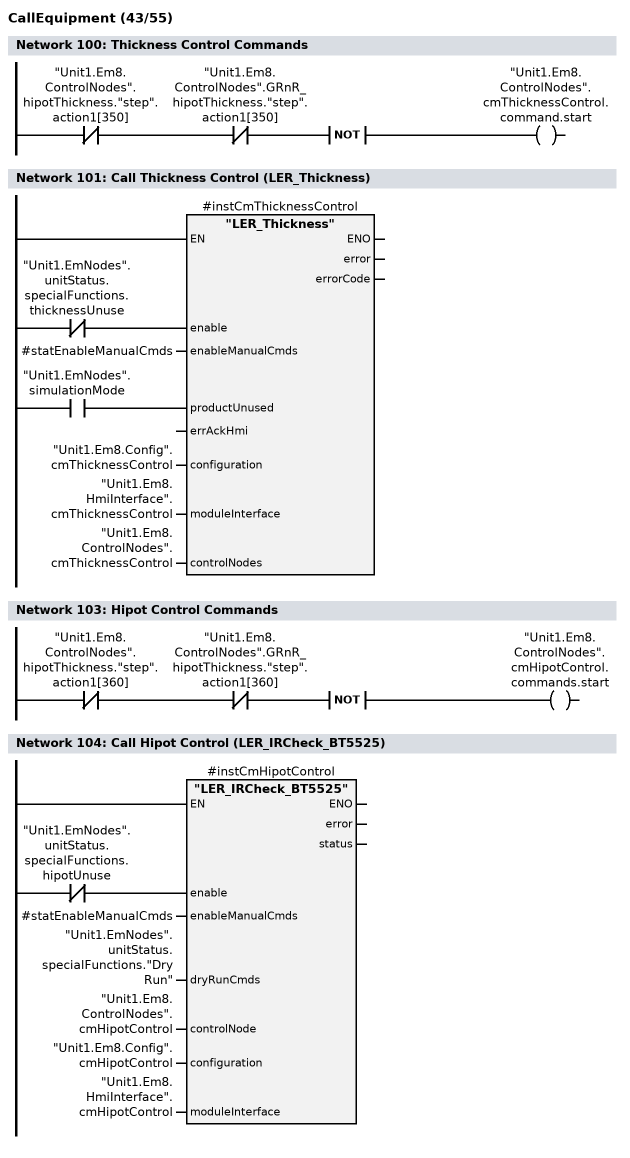
   RUNG wire#powerrail
      I_Contact( "Unit1.Em8.ControlNodes".hipotThickness."step".action1[350] )
      I_Contact( "Unit1.Em8.ControlNodes".GRnR_hipotThickness."step".action1[350] )
      Not()
      Coil( "Unit1.Em8.ControlNodes".cmThicknessControl.command.start )
   END_RUNG
   // the same network as SCL:
   "Unit1.Em8.ControlNodes".cmThicknessControl.command.start := NOT (NOT "Unit1.Em8.ControlNodes".hipotThickness."step".action1[350] AND NOT "Unit1.Em8.ControlNodes".GRnR_hipotThickness."step".action1[350]);
END_REGION

REGION Network 101: Call Thickness Control (LER_Thickness)
   RUNG wire#powerrail
      #instCmThicknessControl(enable := wire#w1, productUnused := wire#w2, enableManualCmds := #statEnableManualCmds, errAckHmi :=, configuration := "Unit1.Em8.Config".cmThicknessControl, moduleInterface := "Unit1.Em8.HmiInterface".cmThicknessControl, controlNodes := "Unit1.Em8.ControlNodes".cmThicknessControl, error =>, errorCode =>)
   END_RUNG
   RUNG wire#powerrail
      I_Contact( "Unit1.EmNodes".unitStatus.specialFunctions.thicknessUnuse )
   END_RUNG wire#w1
   RUNG wire#powerrail
      Contact( "Unit1.EmNodes".simulationMode )
   END_RUNG wire#w2
   // the same network as SCL:
   #instCmThicknessControl(enable := NOT "Unit1.EmNodes".unitStatus.specialFunctions.thicknessUnuse,   // "LER_Thickness"
                           enableManualCmds := #statEnableManualCmds,
                           productUnused := "Unit1.EmNodes".simulationMode,
                           configuration := "Unit1.Em8.Config".cmThicknessControl,
                           moduleInterface := "Unit1.Em8.HmiInterface".cmThicknessControl,
                           controlNodes := "Unit1.Em8.ControlNodes".cmThicknessControl);
END_REGION

REGION Network 103: Hipot Control Commands
   RUNG wire#powerrail
      I_Contact( "Unit1.Em8.ControlNodes".hipotThickness."step".action1[360] )
      I_Contact( "Unit1.Em8.ControlNodes".GRnR_hipotThickness."step".action1[360] )
      Not()
      Coil( "Unit1.Em8.ControlNodes".cmHipotControl.commands.start )
   END_RUNG
   // the same network as SCL:
   "Unit1.Em8.ControlNodes".cmHipotControl.commands.start := NOT (NOT "Unit1.Em8.ControlNodes".hipotThickness."step".action1[360] AND NOT "Unit1.Em8.ControlNodes".GRnR_hipotThickness."step".action1[360]);
END_REGION

REGION Network 104: Call Hipot Control (LER_IRCheck_BT5525)
   RUNG wire#powerrail
      #instCmHipotControl(enable := wire#w1, enableManualCmds := #statEnableManualCmds, dryRunCmds := "Unit1.EmNodes".unitStatus.specialFunctions."Dry Run", controlNode := "Unit1.Em8.ControlNodes".cmHipotControl, configuration := "Unit1.Em8.Config".cmHipotControl, moduleInterface := "Unit1.Em8.HmiInterface".cmHipotControl, error =>, status =>)
   END_RUNG
   RUNG wire#powerrail
      I_Contact( "Unit1.EmNodes".unitStatus.specialFunctions.hipotUnuse )
   END_RUNG wire#w1
   // the same network as SCL:
   #instCmHipotControl(enable := NOT "Unit1.EmNodes".unitStatus.specialFunctions.hipotUnuse,   // "LER_IRCheck_BT5525"
                       enableManualCmds := #statEnableManualCmds,
                       dryRunCmds := "Unit1.EmNodes".unitStatus.specialFunctions."Dry Run",
                       controlNode := "Unit1.Em8.ControlNodes".cmHipotControl,
                       configuration := "Unit1.Em8.Config".cmHipotControl,
                       moduleInterface := "Unit1.Em8.HmiInterface".cmHipotControl);
END_REGION

REGION Network 106: Servo Press Interlock Condition
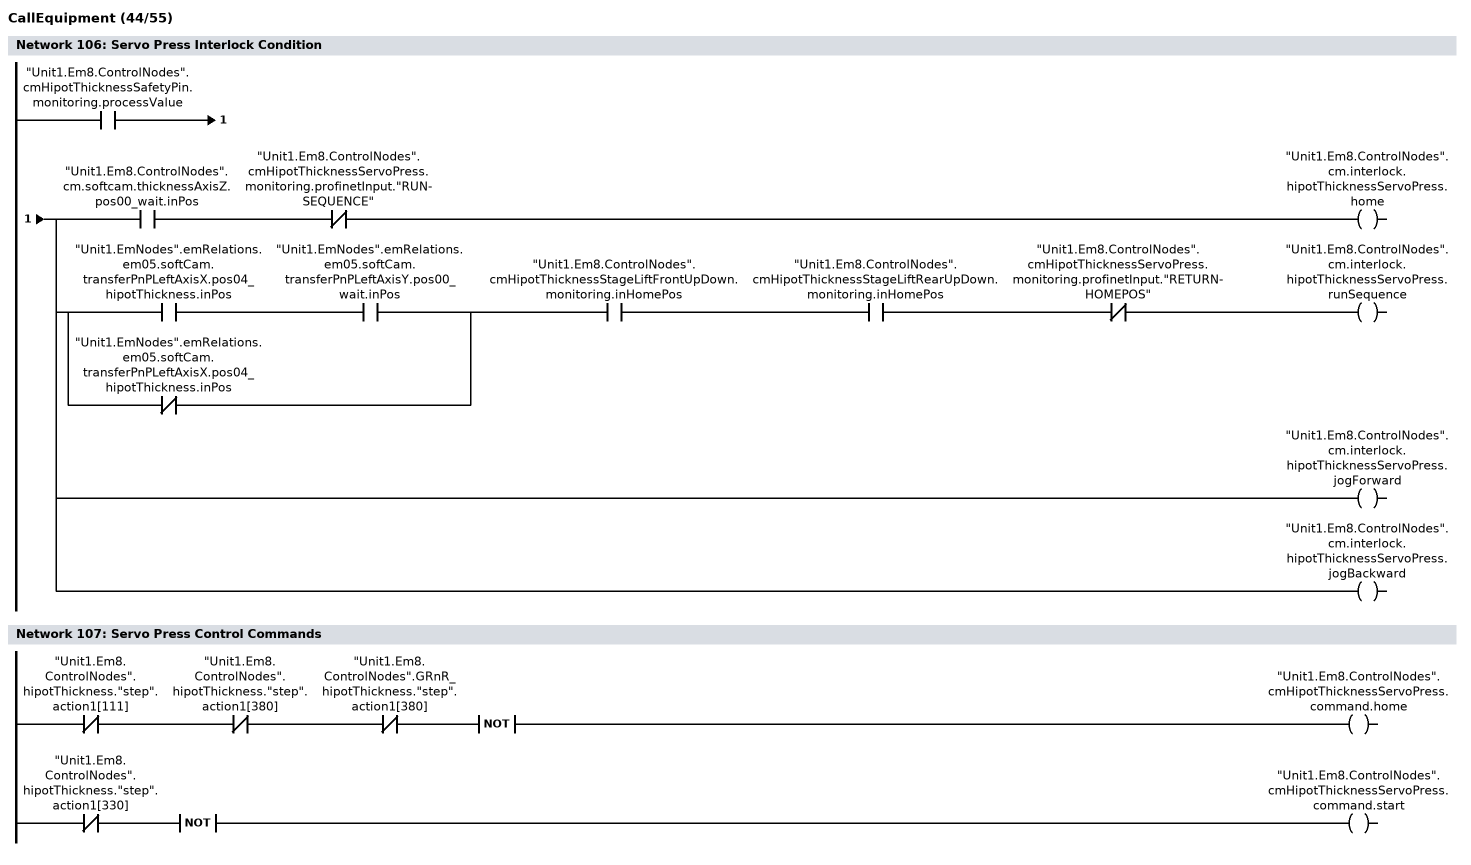
   RUNG wire#powerrail
      Contact( "Unit1.Em8.ControlNodes".cmHipotThicknessSafetyPin.monitoring.processValue )
      wire#w1
      Contact( "Unit1.Em8.ControlNodes".cm.softcam.thicknessAxisZ.pos00_wait.inPos )
      I_Contact( "Unit1.Em8.ControlNodes".cmHipotThicknessServoPress.monitoring.profinetInput."RUN-SEQUENCE" )
      Coil( "Unit1.Em8.ControlNodes".cm.interlock.hipotThicknessServoPress.home )
   END_RUNG
   RUNG wire#w1
      Contact( "Unit1.EmNodes".emRelations.em05.softCam.transferPnPLeftAxisX.pos04_hipotThickness.inPos )
      Contact( "Unit1.EmNodes".emRelations.em05.softCam.transferPnPLeftAxisY.pos00_wait.inPos )
      wire#w2
      Contact( "Unit1.Em8.ControlNodes".cmHipotThicknessStageLiftFrontUpDown.monitoring.inHomePos )
      Contact( "Unit1.Em8.ControlNodes".cmHipotThicknessStageLiftRearUpDown.monitoring.inHomePos )
      I_Contact( "Unit1.Em8.ControlNodes".cmHipotThicknessServoPress.monitoring.profinetInput."RETURN-HOMEPOS" )
      Coil( "Unit1.Em8.ControlNodes".cm.interlock.hipotThicknessServoPress.runSequence )
   END_RUNG
   RUNG wire#w1
      I_Contact( "Unit1.EmNodes".emRelations.em05.softCam.transferPnPLeftAxisX.pos04_hipotThickness.inPos )
   END_RUNG wire#w2
   RUNG wire#w1
      Coil( "Unit1.Em8.ControlNodes".cm.interlock.hipotThicknessServoPress.jogForward )
   END_RUNG
   RUNG wire#w1
      Coil( "Unit1.Em8.ControlNodes".cm.interlock.hipotThicknessServoPress.jogBackward )
   END_RUNG
   // the same network as SCL:
   "Unit1.Em8.ControlNodes".cm.interlock.hipotThicknessServoPress.home := "Unit1.Em8.ControlNodes".cmHipotThicknessSafetyPin.monitoring.processValue AND "Unit1.Em8.ControlNodes".cm.softcam.thicknessAxisZ.pos00_wait.inPos AND NOT "Unit1.Em8.ControlNodes".cmHipotThicknessServoPress.monitoring.profinetInput."RUN-SEQUENCE";
   "Unit1.Em8.ControlNodes".cm.interlock.hipotThicknessServoPress.runSequence := "Unit1.Em8.ControlNodes".cmHipotThicknessSafetyPin.monitoring.processValue AND (("Unit1.EmNodes".emRelations.em05.softCam.transferPnPLeftAxisX.pos04_hipotThickness.inPos AND "Unit1.EmNodes".emRelations.em05.softCam.transferPnPLeftAxisY.pos00_wait.inPos) OR NOT "Unit1.EmNodes".emRelations.em05.softCam.transferPnPLeftAxisX.pos04_hipotThickness.inPos) AND "Unit1.Em8.ControlNodes".cmHipotThicknessStageLiftFrontUpDown.monitoring.inHomePos AND "Unit1.Em8.ControlNodes".cmHipotThicknessStageLiftRearUpDown.monitoring.inHomePos AND NOT "Unit1.Em8.ControlNodes".cmHipotThicknessServoPress.monitoring.profinetInput."RETURN-HOMEPOS";
   "Unit1.Em8.ControlNodes".cm.interlock.hipotThicknessServoPress.jogForward := "Unit1.Em8.ControlNodes".cmHipotThicknessSafetyPin.monitoring.processValue;
   "Unit1.Em8.ControlNodes".cm.interlock.hipotThicknessServoPress.jogBackward := "Unit1.Em8.ControlNodes".cmHipotThicknessSafetyPin.monitoring.processValue;
END_REGION

REGION Network 107: Servo Press Control Commands
   RUNG wire#powerrail
      I_Contact( "Unit1.Em8.ControlNodes".hipotThickness."step".action1[111] )
      I_Contact( "Unit1.Em8.ControlNodes".hipotThickness."step".action1[380] )
      I_Contact( "Unit1.Em8.ControlNodes".GRnR_hipotThickness."step".action1[380] )
      Not()
      Coil( "Unit1.Em8.ControlNodes".cmHipotThicknessServoPress.command.home )
   END_RUNG
   RUNG wire#powerrail
      I_Contact( "Unit1.Em8.ControlNodes".hipotThickness."step".action1[330] )
      Not()
      Coil( "Unit1.Em8.ControlNodes".cmHipotThicknessServoPress.command.start )
   END_RUNG
   // the same network as SCL:
   "Unit1.Em8.ControlNodes".cmHipotThicknessServoPress.command.home := NOT (NOT "Unit1.Em8.ControlNodes".hipotThickness."step".action1[111] AND NOT "Unit1.Em8.ControlNodes".hipotThickness."step".action1[380] AND NOT "Unit1.Em8.ControlNodes".GRnR_hipotThickness."step".action1[380]);
   "Unit1.Em8.ControlNodes".cmHipotThicknessServoPress.command.start := NOT (NOT "Unit1.Em8.ControlNodes".hipotThickness."step".action1[330]);
END_REGION

REGION Network 108: Call CM Servo Press Control
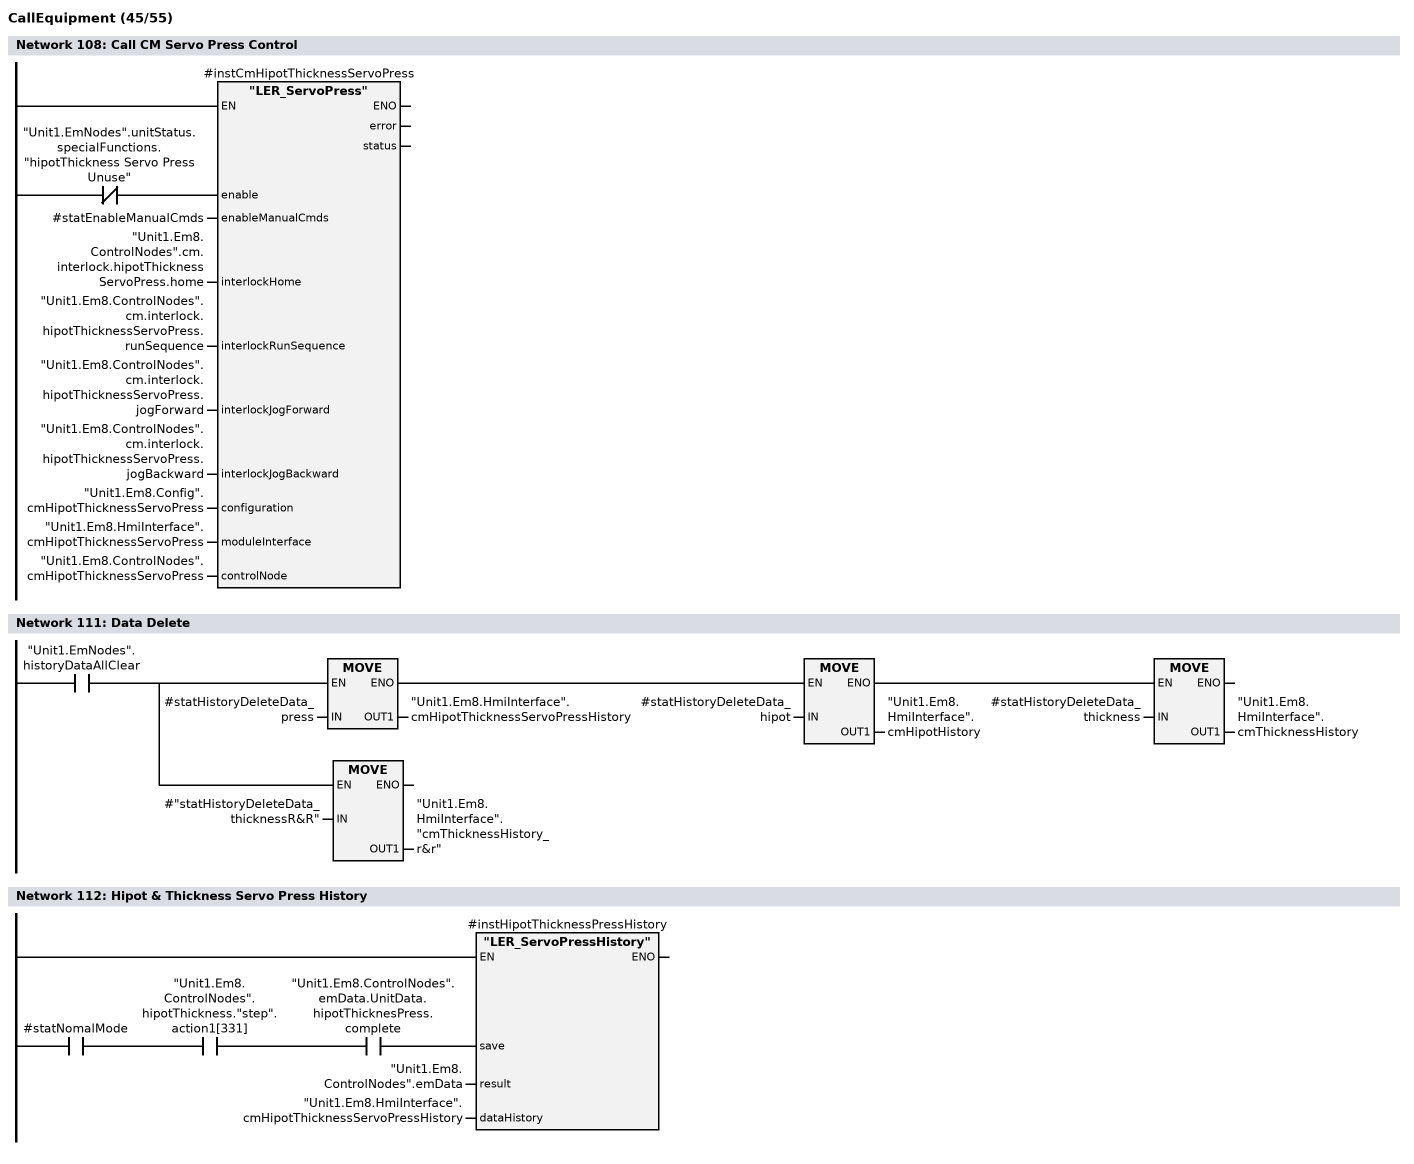
   RUNG wire#powerrail
      #instCmHipotThicknessServoPress(enable := wire#w1, enableManualCmds := #statEnableManualCmds, interlockHome := "Unit1.Em8.ControlNodes".cm.interlock.hipotThicknessServoPress.home, interlockRunSequence := "Unit1.Em8.ControlNodes".cm.interlock.hipotThicknessServoPress.runSequence, interlockJogForward := "Unit1.Em8.ControlNodes".cm.interlock.hipotThicknessServoPress.jogForward, interlockJogBackward := "Unit1.Em8.ControlNodes".cm.interlock.hipotThicknessServoPress.jogBackward, configuration := "Unit1.Em8.Config".cmHipotThicknessServoPress, moduleInterface := "Unit1.Em8.HmiInterface".cmHipotThicknessServoPress, controlNode := "Unit1.Em8.ControlNodes".cmHipotThicknessServoPress, error =>, status =>)
   END_RUNG
   RUNG wire#powerrail
      I_Contact( "Unit1.EmNodes".unitStatus.specialFunctions."hipotThickness Servo Press Unuse" )
   END_RUNG wire#w1
   // the same network as SCL:
   #instCmHipotThicknessServoPress(enable := NOT "Unit1.EmNodes".unitStatus.specialFunctions."hipotThickness Servo Press Unuse",   // "LER_ServoPress"
                           enableManualCmds := #statEnableManualCmds,
                           interlockHome := "Unit1.Em8.ControlNodes".cm.interlock.hipotThicknessServoPress.home,
                           interlockRunSequence := "Unit1.Em8.ControlNodes".cm.interlock.hipotThicknessServoPress.runSequence,
                           interlockJogForward := "Unit1.Em8.ControlNodes".cm.interlock.hipotThicknessServoPress.jogForward,
                           interlockJogBackward := "Unit1.Em8.ControlNodes".cm.interlock.hipotThicknessServoPress.jogBackward,
                           configuration := "Unit1.Em8.Config".cmHipotThicknessServoPress,
                           moduleInterface := "Unit1.Em8.HmiInterface".cmHipotThicknessServoPress,
                           controlNode := "Unit1.Em8.ControlNodes".cmHipotThicknessServoPress);
END_REGION

REGION Network 110: ******************** History ********************
END_REGION

REGION Network 111: Data Delete
   RUNG wire#powerrail
      Contact( "Unit1.EmNodes".historyDataAllClear )
      wire#w1
      Move(in := #statHistoryDeleteData_press, out1 => "Unit1.Em8.HmiInterface".cmHipotThicknessServoPressHistory)
      Move(in := #statHistoryDeleteData_hipot, out1 => "Unit1.Em8.HmiInterface".cmHipotHistory)
      Move(in := #statHistoryDeleteData_thickness, out1 => "Unit1.Em8.HmiInterface".cmThicknessHistory)
   END_RUNG
   RUNG wire#w1
      Move(in := #"statHistoryDeleteData_thicknessR&R", out1 => "Unit1.Em8.HmiInterface"."cmThicknessHistory_r&r")
   END_RUNG
   // the same network as SCL:
   IF "Unit1.EmNodes".historyDataAllClear THEN
       "Unit1.Em8.HmiInterface".cmHipotThicknessServoPressHistory := #statHistoryDeleteData_press;
       "Unit1.Em8.HmiInterface".cmHipotHistory := #statHistoryDeleteData_hipot;
       "Unit1.Em8.HmiInterface".cmThicknessHistory := #statHistoryDeleteData_thickness;
       "Unit1.Em8.HmiInterface"."cmThicknessHistory_r&r" := #"statHistoryDeleteData_thicknessR&R";
   END_IF;
END_REGION

REGION Network 112: Hipot & Thickness Servo Press History
   RUNG wire#powerrail
      #instHipotThicknessPressHistory(save := wire#w1, result := "Unit1.Em8.ControlNodes".emData, dataHistory := "Unit1.Em8.HmiInterface".cmHipotThicknessServoPressHistory)
   END_RUNG
   RUNG wire#powerrail
      Contact( #statNomalMode )
      Contact( "Unit1.Em8.ControlNodes".hipotThickness."step".action1[331] )
      Contact( "Unit1.Em8.ControlNodes".emData.UnitData.hipotThicknesPress.complete )
   END_RUNG wire#w1
   // the same network as SCL:
   #instHipotThicknessPressHistory(save := #statNomalMode AND "Unit1.Em8.ControlNodes".hipotThickness."step".action1[331] AND "Unit1.Em8.ControlNodes".emData.UnitData.hipotThicknesPress.complete,   // "LER_ServoPressHistory"
                           result := "Unit1.Em8.ControlNodes".emData,
                           dataHistory := "Unit1.Em8.HmiInterface".cmHipotThicknessServoPressHistory);
END_REGION

REGION Network 113: Hipot History
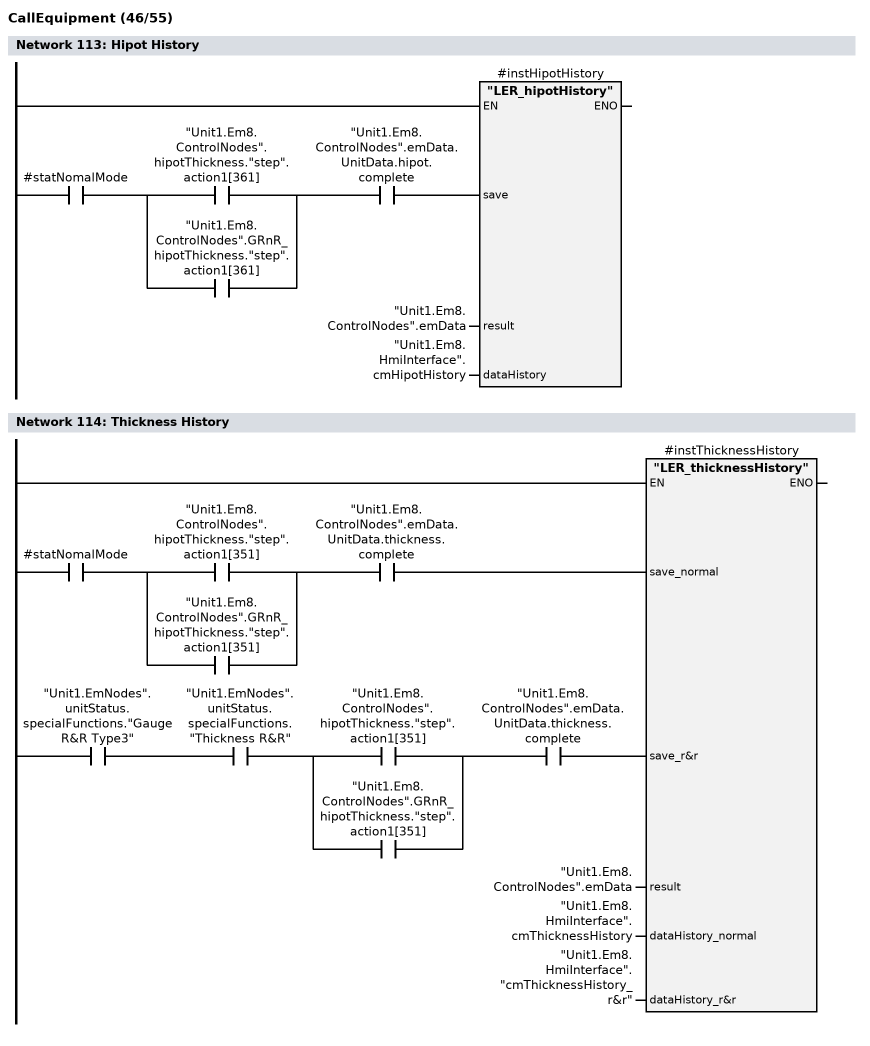
   RUNG wire#powerrail
      #instHipotHistory(save := wire#w3, result := "Unit1.Em8.ControlNodes".emData, dataHistory := "Unit1.Em8.HmiInterface".cmHipotHistory)
   END_RUNG
   RUNG wire#powerrail
      Contact( #statNomalMode )
      wire#w1
      Contact( "Unit1.Em8.ControlNodes".hipotThickness."step".action1[361] )
      wire#w2
      Contact( "Unit1.Em8.ControlNodes".emData.UnitData.hipot.complete )
   END_RUNG wire#w3
   RUNG wire#w1
      Contact( "Unit1.Em8.ControlNodes".GRnR_hipotThickness."step".action1[361] )
   END_RUNG wire#w2
   // the same network as SCL:
   #instHipotHistory(save := #statNomalMode AND ("Unit1.Em8.ControlNodes".hipotThickness."step".action1[361] OR "Unit1.Em8.ControlNodes".GRnR_hipotThickness."step".action1[361]) AND "Unit1.Em8.ControlNodes".emData.UnitData.hipot.complete,   // "LER_hipotHistory"
                     result := "Unit1.Em8.ControlNodes".emData,
                     dataHistory := "Unit1.Em8.HmiInterface".cmHipotHistory);
END_REGION

REGION Network 114: Thickness History
   RUNG wire#powerrail
      #instThicknessHistory(save_normal := wire#w3, "save_r&r" := wire#w6, result := "Unit1.Em8.ControlNodes".emData, dataHistory_normal := "Unit1.Em8.HmiInterface".cmThicknessHistory, "dataHistory_r&r" := "Unit1.Em8.HmiInterface"."cmThicknessHistory_r&r")
   END_RUNG
   RUNG wire#powerrail
      Contact( #statNomalMode )
      wire#w1
      Contact( "Unit1.Em8.ControlNodes".hipotThickness."step".action1[351] )
      wire#w2
      Contact( "Unit1.Em8.ControlNodes".emData.UnitData.thickness.complete )
   END_RUNG wire#w3
   RUNG wire#w1
      Contact( "Unit1.Em8.ControlNodes".GRnR_hipotThickness."step".action1[351] )
   END_RUNG wire#w2
   RUNG wire#powerrail
      Contact( "Unit1.EmNodes".unitStatus.specialFunctions."Gauge R&R Type3" )
      Contact( "Unit1.EmNodes".unitStatus.specialFunctions."Thickness R&R" )
      wire#w4
      Contact( "Unit1.Em8.ControlNodes".hipotThickness."step".action1[351] )
      wire#w5
      Contact( "Unit1.Em8.ControlNodes".emData.UnitData.thickness.complete )
   END_RUNG wire#w6
   RUNG wire#w4
      Contact( "Unit1.Em8.ControlNodes".GRnR_hipotThickness."step".action1[351] )
   END_RUNG wire#w5
   // the same network as SCL:
   #instThicknessHistory(save_normal := #statNomalMode AND ("Unit1.Em8.ControlNodes".hipotThickness."step".action1[351] OR "Unit1.Em8.ControlNodes".GRnR_hipotThickness."step".action1[351]) AND "Unit1.Em8.ControlNodes".emData.UnitData.thickness.complete,   // "LER_thicknessHistory"
                         "save_r&r" := "Unit1.EmNodes".unitStatus.specialFunctions."Gauge R&R Type3" AND "Unit1.EmNodes".unitStatus.specialFunctions."Thickness R&R" AND ("Unit1.Em8.ControlNodes".hipotThickness."step".action1[351] OR "Unit1.Em8.ControlNodes".GRnR_hipotThickness."step".action1[351]) AND "Unit1.Em8.ControlNodes".emData.UnitData.thickness.complete,
                         result := "Unit1.Em8.ControlNodes".emData,
                         dataHistory_normal := "Unit1.Em8.HmiInterface".cmThicknessHistory,
                         "dataHistory_r&r" := "Unit1.Em8.HmiInterface"."cmThicknessHistory_r&r");
END_REGION

REGION Network 116: ******************** Feedback to Unit ********************
END_REGION

REGION Network 117: Determine StateComplete (SC) in Mode Production
   // Conditions for the Equipment Modules "stateComplete" feedback to the unit. This feedback is given when the task in for the respective state is complete.
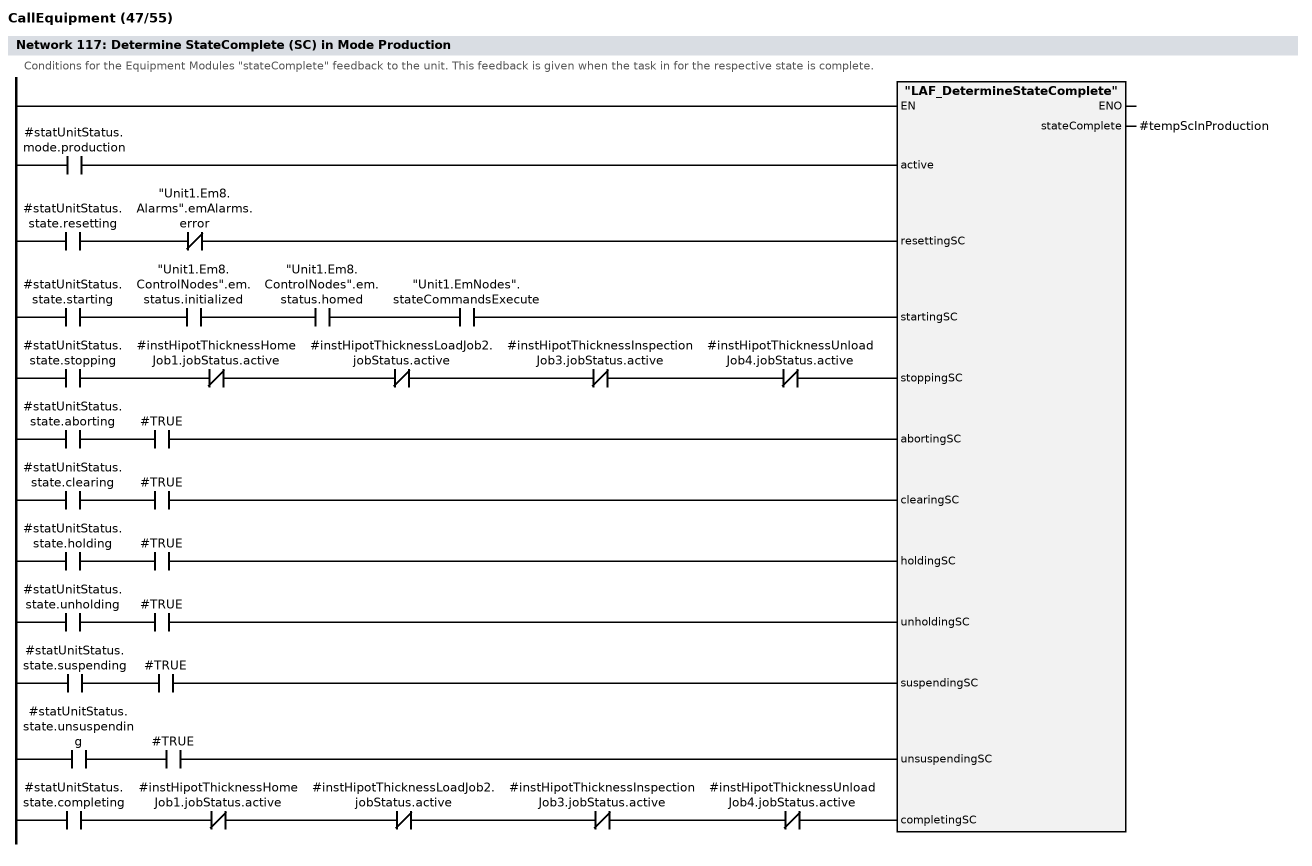
   RUNG wire#powerrail
      "LAF_DetermineStateComplete"(active := wire#w1, resettingSC := wire#w2, startingSC := wire#w3, stoppingSC := wire#w4, abortingSC := wire#w5, clearingSC := wire#w6, holdingSC := wire#w7, unholdingSC := wire#w8, suspendingSC := wire#w9, unsuspendingSC := wire#w10, completingSC := wire#w11, stateComplete => #tempScInProduction)
   END_RUNG
   RUNG wire#powerrail
      Contact( #statUnitStatus.mode.production )
   END_RUNG wire#w1
   RUNG wire#powerrail
      Contact( #statUnitStatus.state.resetting )
      I_Contact( "Unit1.Em8.Alarms".emAlarms.error )
   END_RUNG wire#w2
   RUNG wire#powerrail
      Contact( #statUnitStatus.state.starting )
      Contact( "Unit1.Em8.ControlNodes".em.status.initialized )
      Contact( "Unit1.Em8.ControlNodes".em.status.homed )
      Contact( "Unit1.EmNodes".stateCommandsExecute )
   END_RUNG wire#w3
   RUNG wire#powerrail
      Contact( #statUnitStatus.state.stopping )
      I_Contact( #instHipotThicknessHomeJob1.jobStatus.active )
      I_Contact( #instHipotThicknessLoadJob2.jobStatus.active )
      I_Contact( #instHipotThicknessInspectionJob3.jobStatus.active )
      I_Contact( #instHipotThicknessUnloadJob4.jobStatus.active )
   END_RUNG wire#w4
   RUNG wire#powerrail
      Contact( #statUnitStatus.state.aborting )
      Contact( #TRUE )
   END_RUNG wire#w5
   RUNG wire#powerrail
      Contact( #statUnitStatus.state.clearing )
      Contact( #TRUE )
   END_RUNG wire#w6
   RUNG wire#powerrail
      Contact( #statUnitStatus.state.holding )
      Contact( #TRUE )
   END_RUNG wire#w7
   RUNG wire#powerrail
      Contact( #statUnitStatus.state.unholding )
      Contact( #TRUE )
   END_RUNG wire#w8
   RUNG wire#powerrail
      Contact( #statUnitStatus.state.suspending )
      Contact( #TRUE )
   END_RUNG wire#w9
   RUNG wire#powerrail
      Contact( #statUnitStatus.state.unsuspending )
      Contact( #TRUE )
   END_RUNG wire#w10
   RUNG wire#powerrail
      Contact( #statUnitStatus.state.completing )
      I_Contact( #instHipotThicknessHomeJob1.jobStatus.active )
      I_Contact( #instHipotThicknessLoadJob2.jobStatus.active )
      I_Contact( #instHipotThicknessInspectionJob3.jobStatus.active )
      I_Contact( #instHipotThicknessUnloadJob4.jobStatus.active )
   END_RUNG wire#w11
   // the same network as SCL:
   "LAF_DetermineStateComplete"(active := #statUnitStatus.mode.production,
                           resettingSC := #statUnitStatus.state.resetting AND NOT "Unit1.Em8.Alarms".emAlarms.error,
                           startingSC := #statUnitStatus.state.starting AND "Unit1.Em8.ControlNodes".em.status.initialized AND "Unit1.Em8.ControlNodes".em.status.homed AND "Unit1.EmNodes".stateCommandsExecute,
                           stoppingSC := #statUnitStatus.state.stopping AND NOT #instHipotThicknessHomeJob1.jobStatus.active AND NOT #instHipotThicknessLoadJob2.jobStatus.active AND NOT #instHipotThicknessInspectionJob3.jobStatus.active AND NOT #instHipotThicknessUnloadJob4.jobStatus.active,
                           abortingSC := #statUnitStatus.state.aborting AND #TRUE,
                           clearingSC := #statUnitStatus.state.clearing AND #TRUE,
                           holdingSC := #statUnitStatus.state.holding AND #TRUE,
                           unholdingSC := #statUnitStatus.state.unholding AND #TRUE,
                           suspendingSC := #statUnitStatus.state.suspending AND #TRUE,
                           unsuspendingSC := #statUnitStatus.state.unsuspending AND #TRUE,
                           completingSC := #statUnitStatus.state.completing AND NOT #instHipotThicknessHomeJob1.jobStatus.active AND NOT #instHipotThicknessLoadJob2.jobStatus.active AND NOT #instHipotThicknessInspectionJob3.jobStatus.active AND NOT #instHipotThicknessUnloadJob4.jobStatus.active,
                           stateComplete => #tempScInProduction);
END_REGION

REGION Network 118: Determine StateComplete (SC) in Mode Maintenance/Manual
   // Conditions for the Equipment Modules "stateComplete" feedback to the unit. This feedback is given when the task in for the respective state is complete.
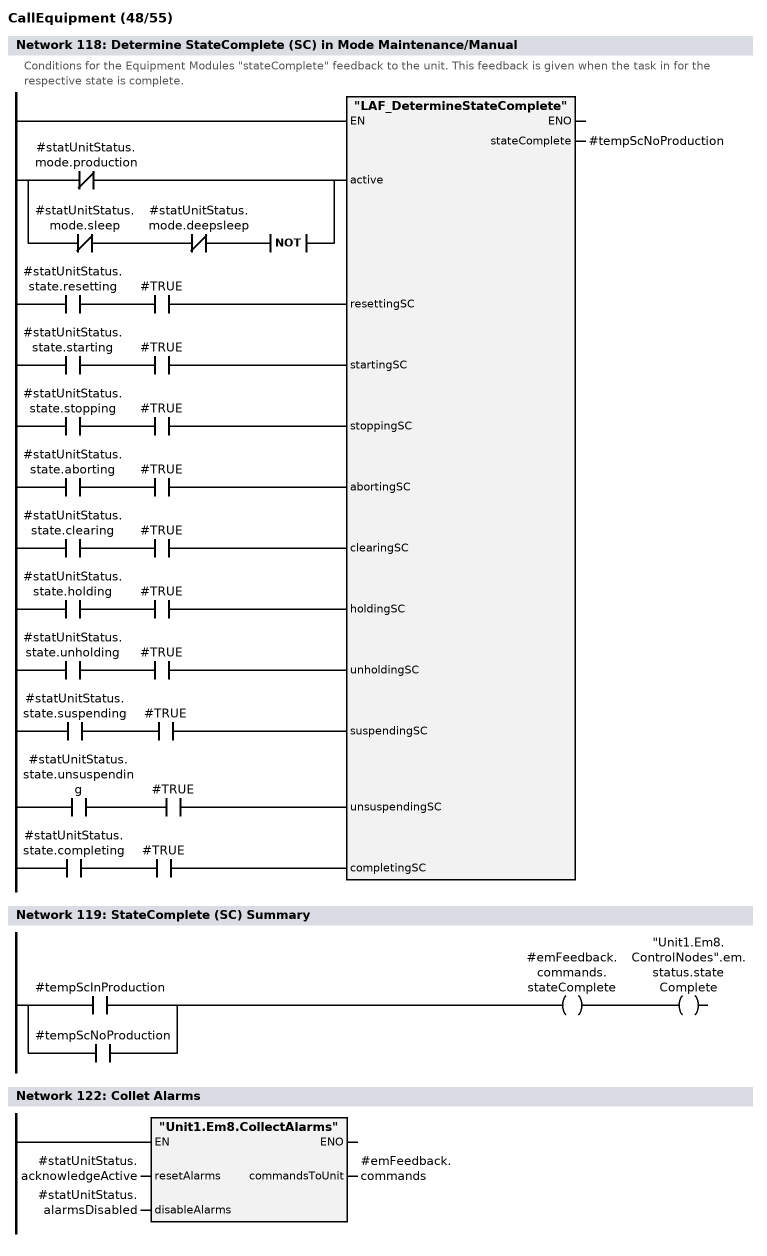
   RUNG wire#powerrail
      "LAF_DetermineStateComplete"(active := wire#w1, resettingSC := wire#w2, startingSC := wire#w3, stoppingSC := wire#w4, abortingSC := wire#w5, clearingSC := wire#w6, holdingSC := wire#w7, unholdingSC := wire#w8, suspendingSC := wire#w9, unsuspendingSC := wire#w10, completingSC := wire#w11, stateComplete => #tempScNoProduction)
   END_RUNG
   RUNG wire#powerrail
      I_Contact( #statUnitStatus.mode.production )
   END_RUNG wire#w1
   RUNG wire#powerrail
      I_Contact( #statUnitStatus.mode.sleep )
      I_Contact( #statUnitStatus.mode.deepsleep )
      Not()
   END_RUNG wire#w1
   RUNG wire#powerrail
      Contact( #statUnitStatus.state.resetting )
      Contact( #TRUE )
   END_RUNG wire#w2
   RUNG wire#powerrail
      Contact( #statUnitStatus.state.starting )
      Contact( #TRUE )
   END_RUNG wire#w3
   RUNG wire#powerrail
      Contact( #statUnitStatus.state.stopping )
      Contact( #TRUE )
   END_RUNG wire#w4
   RUNG wire#powerrail
      Contact( #statUnitStatus.state.aborting )
      Contact( #TRUE )
   END_RUNG wire#w5
   RUNG wire#powerrail
      Contact( #statUnitStatus.state.clearing )
      Contact( #TRUE )
   END_RUNG wire#w6
   RUNG wire#powerrail
      Contact( #statUnitStatus.state.holding )
      Contact( #TRUE )
   END_RUNG wire#w7
   RUNG wire#powerrail
      Contact( #statUnitStatus.state.unholding )
      Contact( #TRUE )
   END_RUNG wire#w8
   RUNG wire#powerrail
      Contact( #statUnitStatus.state.suspending )
      Contact( #TRUE )
   END_RUNG wire#w9
   RUNG wire#powerrail
      Contact( #statUnitStatus.state.unsuspending )
      Contact( #TRUE )
   END_RUNG wire#w10
   RUNG wire#powerrail
      Contact( #statUnitStatus.state.completing )
      Contact( #TRUE )
   END_RUNG wire#w11
   // the same network as SCL:
   "LAF_DetermineStateComplete"(active := NOT #statUnitStatus.mode.production OR NOT (NOT #statUnitStatus.mode.sleep AND NOT #statUnitStatus.mode.deepsleep),
                           resettingSC := #statUnitStatus.state.resetting AND #TRUE,
                           startingSC := #statUnitStatus.state.starting AND #TRUE,
                           stoppingSC := #statUnitStatus.state.stopping AND #TRUE,
                           abortingSC := #statUnitStatus.state.aborting AND #TRUE,
                           clearingSC := #statUnitStatus.state.clearing AND #TRUE,
                           holdingSC := #statUnitStatus.state.holding AND #TRUE,
                           unholdingSC := #statUnitStatus.state.unholding AND #TRUE,
                           suspendingSC := #statUnitStatus.state.suspending AND #TRUE,
                           unsuspendingSC := #statUnitStatus.state.unsuspending AND #TRUE,
                           completingSC := #statUnitStatus.state.completing AND #TRUE,
                           stateComplete => #tempScNoProduction);
END_REGION

REGION Network 119: StateComplete (SC) Summary
   RUNG wire#powerrail
      Contact( #tempScInProduction )
      wire#w1
      Coil( #emFeedback.commands.stateComplete )
      Coil( "Unit1.Em8.ControlNodes".em.status.stateComplete )
   END_RUNG
   RUNG wire#powerrail
      Contact( #tempScNoProduction )
   END_RUNG wire#w1
   // the same network as SCL:
   #emFeedback.commands.stateComplete := #tempScInProduction OR #tempScNoProduction;
   "Unit1.Em8.ControlNodes".em.status.stateComplete := #emFeedback.commands.stateComplete;
END_REGION

REGION Network 121: ******************** Alarms ********************
END_REGION

REGION Network 122: Collet Alarms
   RUNG wire#powerrail
      "Unit1.Em8.CollectAlarms"(resetAlarms := #statUnitStatus.acknowledgeActive, disableAlarms := #statUnitStatus.alarmsDisabled, commandsToUnit => #emFeedback.commands)
   END_RUNG
   // the same network as SCL:
   "Unit1.Em8.CollectAlarms"(resetAlarms := #statUnitStatus.acknowledgeActive,
                           disableAlarms := #statUnitStatus.alarmsDisabled,
                           commandsToUnit => #emFeedback.commands);
END_REGION

REGION Network 123: Manage Alarms
   // Derive commands from the ProDiag supervision. The ProDiag supervisions contain categories which define the reaction of these supervisions (e.g. abort, stop, hold). These are handed over as commands to the unit level.
   // Alternatively, if no ProDiag should be used, you can use the LAF_ManageBitAlarms to realize bit alarm handling. This block can be found in LAF in folder 70_AlarmHandling.
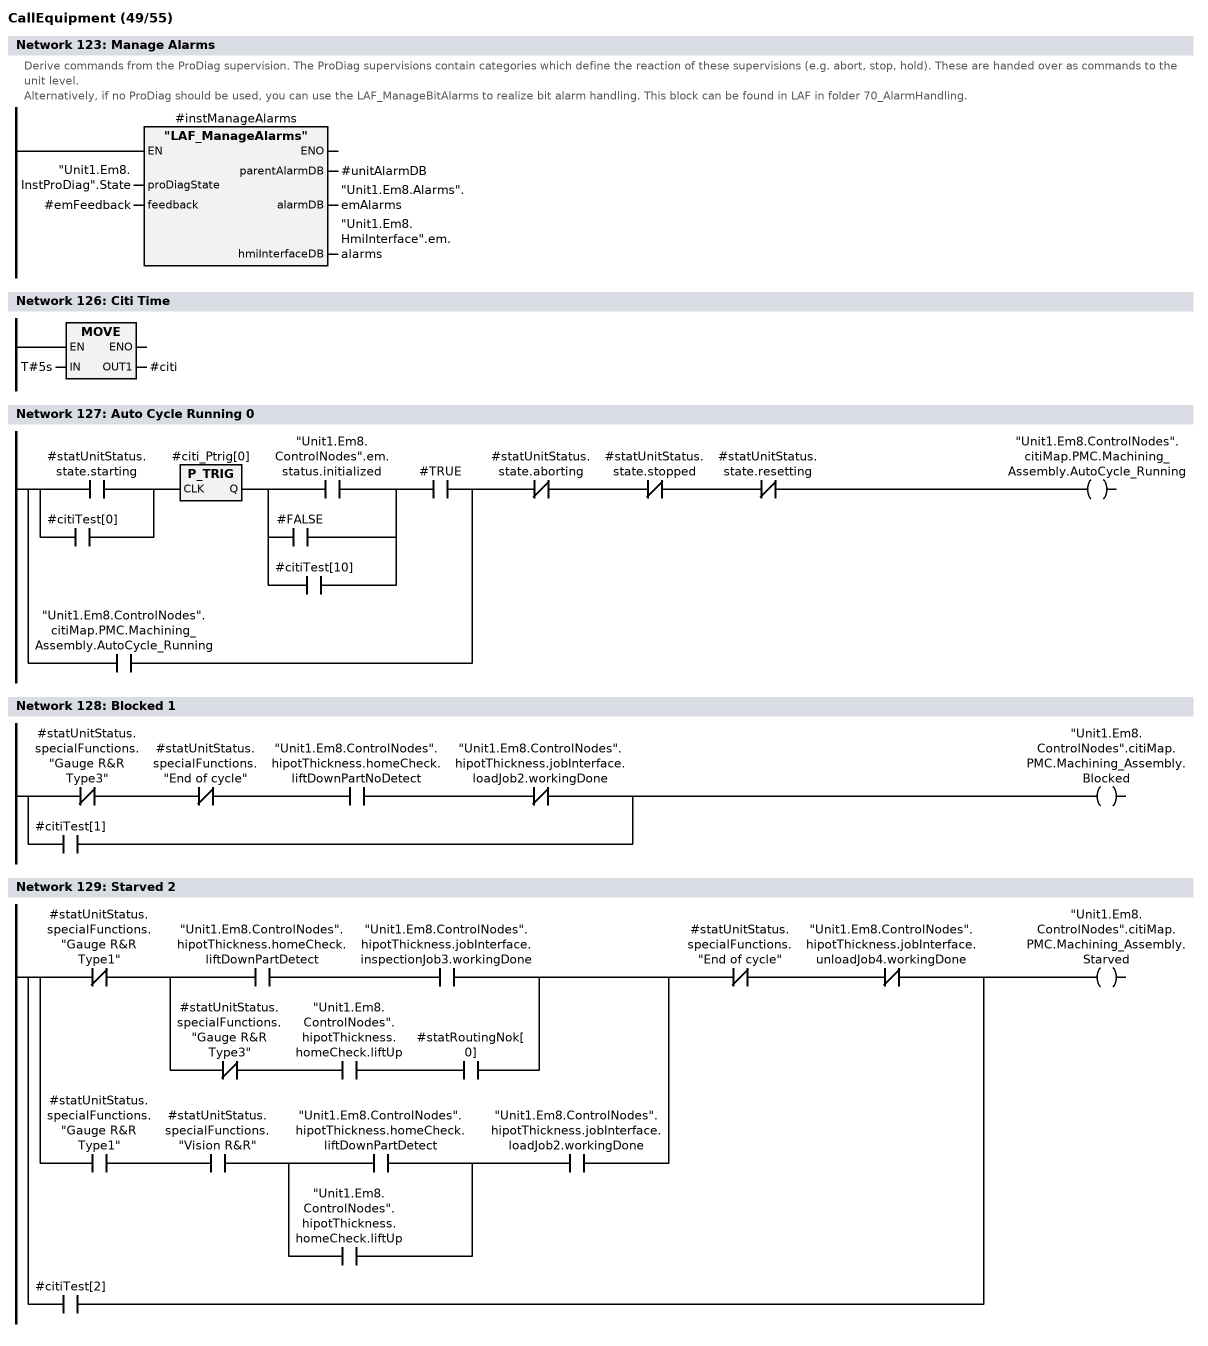
   RUNG wire#powerrail
      #instManageAlarms(proDiagState := "Unit1.Em8.InstProDiag".State, feedback := #emFeedback, parentAlarmDB => #unitAlarmDB, alarmDB => "Unit1.Em8.Alarms".emAlarms, hmiInterfaceDB => "Unit1.Em8.HmiInterface".em.alarms)
   END_RUNG
   // the same network as SCL:
   #instManageAlarms(proDiagState := "Unit1.Em8.InstProDiag".State,   // "LAF_ManageAlarms"
                     feedback := #emFeedback,
                     parentAlarmDB => #unitAlarmDB,
                     alarmDB => "Unit1.Em8.Alarms".emAlarms,
                     hmiInterfaceDB => "Unit1.Em8.HmiInterface".em.alarms);
END_REGION

REGION Network 125: ******************** CITI ********************
END_REGION

REGION Network 126: Citi Time
   RUNG wire#powerrail
      Move(in := T#5s, out1 => #citi)
   END_RUNG
   // the same network as SCL:
   #citi := T#5s;
END_REGION

REGION Network 127: Auto Cycle Running 0
   RUNG wire#powerrail
      Contact( #statUnitStatus.state.starting )
      wire#w1
      P_Trig( #citi_Ptrig[0] )
      wire#w2
      Contact( "Unit1.Em8.ControlNodes".em.status.initialized )
      wire#w3
      Contact( #TRUE )
      wire#w4
      I_Contact( #statUnitStatus.state.aborting )
      I_Contact( #statUnitStatus.state.stopped )
      I_Contact( #statUnitStatus.state.resetting )
      Coil( "Unit1.Em8.ControlNodes".citiMap.PMC.Machining_Assembly.AutoCycle_Running )
   END_RUNG
   RUNG wire#powerrail
      Contact( #citiTest[0] )
   END_RUNG wire#w1
   RUNG wire#w2
      Contact( #FALSE )
   END_RUNG wire#w3
   RUNG wire#w2
      Contact( #citiTest[10] )
   END_RUNG wire#w3
   RUNG wire#powerrail
      Contact( "Unit1.Em8.ControlNodes".citiMap.PMC.Machining_Assembly.AutoCycle_Running )
   END_RUNG wire#w4
   // the same network as SCL:
   #_w1 := #statUnitStatus.state.starting OR #citiTest[0];
   #_w2 := #_w1 AND NOT #citi_Ptrig[0];   // rising edge
   #citi_Ptrig[0] := #_w1;
   "Unit1.Em8.ControlNodes".citiMap.PMC.Machining_Assembly.AutoCycle_Running := ((#_w2 AND ("Unit1.Em8.ControlNodes".em.status.initialized OR #FALSE OR #citiTest[10]) AND #TRUE) OR "Unit1.Em8.ControlNodes".citiMap.PMC.Machining_Assembly.AutoCycle_Running) AND NOT #statUnitStatus.state.aborting AND NOT #statUnitStatus.state.stopped AND NOT #statUnitStatus.state.resetting;
END_REGION

REGION Network 128: Blocked 1
   RUNG wire#powerrail
      I_Contact( #statUnitStatus.specialFunctions."Gauge R&R Type3" )
      I_Contact( #statUnitStatus.specialFunctions."End of cycle" )
      Contact( "Unit1.Em8.ControlNodes".hipotThickness.homeCheck.liftDownPartNoDetect )
      I_Contact( "Unit1.Em8.ControlNodes".hipotThickness.jobInterface.loadJob2.workingDone )
      wire#w1
      Coil( "Unit1.Em8.ControlNodes".citiMap.PMC.Machining_Assembly.Blocked )
   END_RUNG
   RUNG wire#powerrail
      Contact( #citiTest[1] )
   END_RUNG wire#w1
   // the same network as SCL:
   "Unit1.Em8.ControlNodes".citiMap.PMC.Machining_Assembly.Blocked := (NOT #statUnitStatus.specialFunctions."Gauge R&R Type3" AND NOT #statUnitStatus.specialFunctions."End of cycle" AND "Unit1.Em8.ControlNodes".hipotThickness.homeCheck.liftDownPartNoDetect AND NOT "Unit1.Em8.ControlNodes".hipotThickness.jobInterface.loadJob2.workingDone) OR #citiTest[1];
END_REGION

REGION Network 129: Starved 2
   RUNG wire#powerrail
      I_Contact( #statUnitStatus.specialFunctions."Gauge R&R Type1" )
      wire#w1
      Contact( "Unit1.Em8.ControlNodes".hipotThickness.homeCheck.liftDownPartDetect )
      Contact( "Unit1.Em8.ControlNodes".hipotThickness.jobInterface.inspectionJob3.workingDone )
      wire#w2
      I_Contact( #statUnitStatus.specialFunctions."End of cycle" )
      I_Contact( "Unit1.Em8.ControlNodes".hipotThickness.jobInterface.unloadJob4.workingDone )
      wire#w5
      Coil( "Unit1.Em8.ControlNodes".citiMap.PMC.Machining_Assembly.Starved )
   END_RUNG
   RUNG wire#w1
      I_Contact( #statUnitStatus.specialFunctions."Gauge R&R Type3" )
      Contact( "Unit1.Em8.ControlNodes".hipotThickness.homeCheck.liftUp )
      Contact( #statRoutingNok[0] )
   END_RUNG wire#w2
   RUNG wire#powerrail
      Contact( #statUnitStatus.specialFunctions."Gauge R&R Type1" )
      Contact( #statUnitStatus.specialFunctions."Vision R&R" )
      wire#w3
      Contact( "Unit1.Em8.ControlNodes".hipotThickness.homeCheck.liftDownPartDetect )
      wire#w4
      Contact( "Unit1.Em8.ControlNodes".hipotThickness.jobInterface.loadJob2.workingDone )
   END_RUNG wire#w2
   RUNG wire#w3
      Contact( "Unit1.Em8.ControlNodes".hipotThickness.homeCheck.liftUp )
   END_RUNG wire#w4
   RUNG wire#powerrail
      Contact( #citiTest[2] )
   END_RUNG wire#w5
   // the same network as SCL:
   "Unit1.Em8.ControlNodes".citiMap.PMC.Machining_Assembly.Starved := (((NOT #statUnitStatus.specialFunctions."Gauge R&R Type1" AND (("Unit1.Em8.ControlNodes".hipotThickness.homeCheck.liftDownPartDetect AND "Unit1.Em8.ControlNodes".hipotThickness.jobInterface.inspectionJob3.workingDone) OR (NOT #statUnitStatus.specialFunctions."Gauge R&R Type3" AND "Unit1.Em8.ControlNodes".hipotThickness.homeCheck.liftUp AND #statRoutingNok[0]))) OR (#statUnitStatus.specialFunctions."Gauge R&R Type1" AND #statUnitStatus.specialFunctions."Vision R&R" AND ("Unit1.Em8.ControlNodes".hipotThickness.homeCheck.liftDownPartDetect OR "Unit1.Em8.ControlNodes".hipotThickness.homeCheck.liftUp) AND "Unit1.Em8.ControlNodes".hipotThickness.jobInterface.loadJob2.workingDone)) AND NOT #statUnitStatus.specialFunctions."End of cycle" AND NOT "Unit1.Em8.ControlNodes".hipotThickness.jobInterface.unloadJob4.workingDone) OR #citiTest[2];
END_REGION

REGION Network 130: Good Count 3
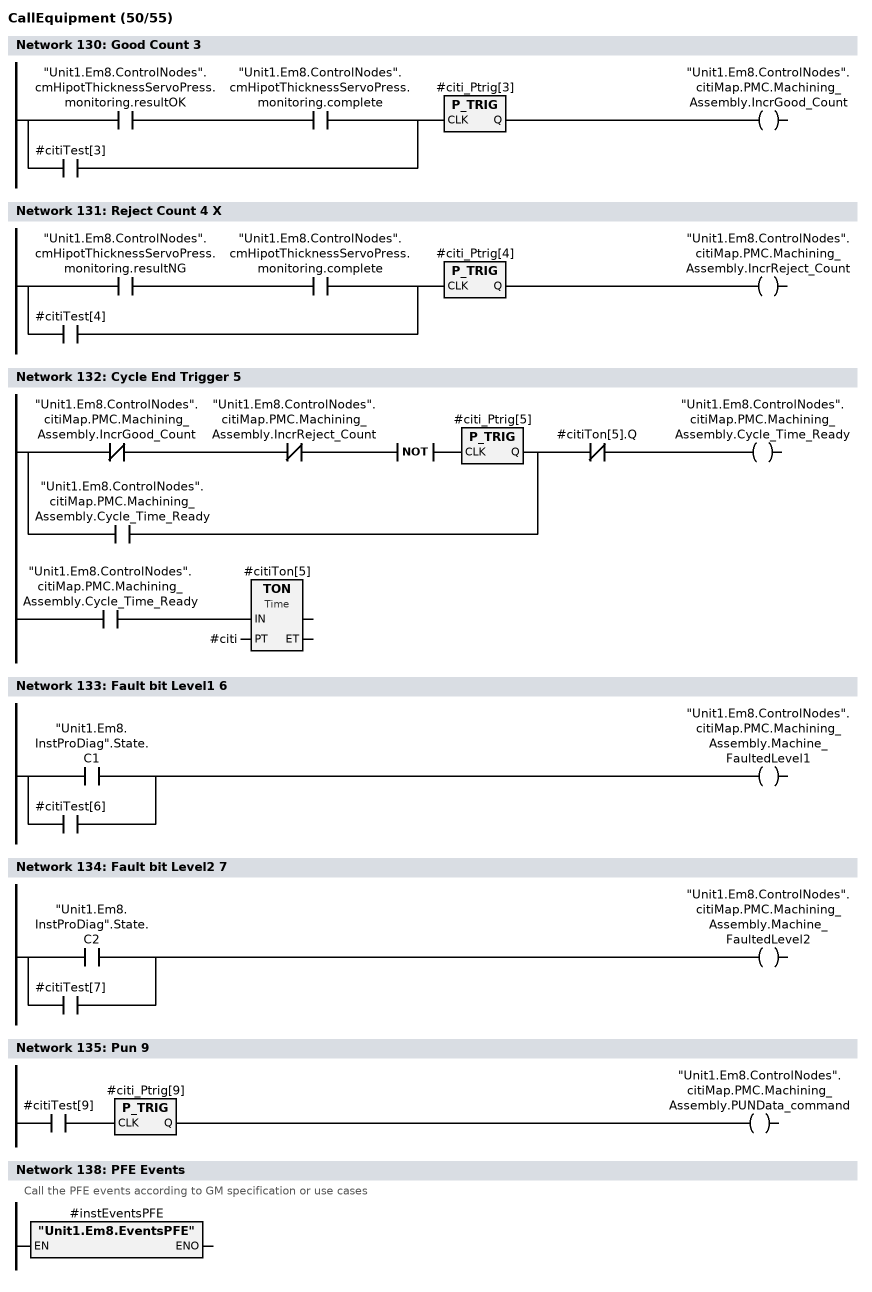
   RUNG wire#powerrail
      Contact( "Unit1.Em8.ControlNodes".cmHipotThicknessServoPress.monitoring.resultOK )
      Contact( "Unit1.Em8.ControlNodes".cmHipotThicknessServoPress.monitoring.complete )
      wire#w1
      P_Trig( #citi_Ptrig[3] )
      Coil( "Unit1.Em8.ControlNodes".citiMap.PMC.Machining_Assembly.IncrGood_Count )
   END_RUNG
   RUNG wire#powerrail
      Contact( #citiTest[3] )
   END_RUNG wire#w1
   // the same network as SCL:
   #_w1 := ("Unit1.Em8.ControlNodes".cmHipotThicknessServoPress.monitoring.resultOK AND "Unit1.Em8.ControlNodes".cmHipotThicknessServoPress.monitoring.complete) OR #citiTest[3];
   #_w2 := #_w1 AND NOT #citi_Ptrig[3];   // rising edge
   #citi_Ptrig[3] := #_w1;
   "Unit1.Em8.ControlNodes".citiMap.PMC.Machining_Assembly.IncrGood_Count := #_w2;
END_REGION

REGION Network 131: Reject Count 4 X
   RUNG wire#powerrail
      Contact( "Unit1.Em8.ControlNodes".cmHipotThicknessServoPress.monitoring.resultNG )
      Contact( "Unit1.Em8.ControlNodes".cmHipotThicknessServoPress.monitoring.complete )
      wire#w1
      P_Trig( #citi_Ptrig[4] )
      Coil( "Unit1.Em8.ControlNodes".citiMap.PMC.Machining_Assembly.IncrReject_Count )
   END_RUNG
   RUNG wire#powerrail
      Contact( #citiTest[4] )
   END_RUNG wire#w1
   // the same network as SCL:
   #_w1 := ("Unit1.Em8.ControlNodes".cmHipotThicknessServoPress.monitoring.resultNG AND "Unit1.Em8.ControlNodes".cmHipotThicknessServoPress.monitoring.complete) OR #citiTest[4];
   #_w2 := #_w1 AND NOT #citi_Ptrig[4];   // rising edge
   #citi_Ptrig[4] := #_w1;
   "Unit1.Em8.ControlNodes".citiMap.PMC.Machining_Assembly.IncrReject_Count := #_w2;
END_REGION

REGION Network 132: Cycle End Trigger 5
   RUNG wire#powerrail
      I_Contact( "Unit1.Em8.ControlNodes".citiMap.PMC.Machining_Assembly.IncrGood_Count )
      I_Contact( "Unit1.Em8.ControlNodes".citiMap.PMC.Machining_Assembly.IncrReject_Count )
      Not()
      P_Trig( #citi_Ptrig[5] )
      wire#w1
      I_Contact( #citiTon[5].Q )
      Coil( "Unit1.Em8.ControlNodes".citiMap.PMC.Machining_Assembly.Cycle_Time_Ready )
   END_RUNG
   RUNG wire#powerrail
      Contact( "Unit1.Em8.ControlNodes".citiMap.PMC.Machining_Assembly.Cycle_Time_Ready )
   END_RUNG wire#w1
   RUNG wire#powerrail
      Contact( "Unit1.Em8.ControlNodes".citiMap.PMC.Machining_Assembly.Cycle_Time_Ready )
      { S7_Templates := "time_type := Time" } #citiTon[5].TON(pt := #citi, et =>)
   END_RUNG
   // the same network as SCL:
   #_w1 := NOT (NOT "Unit1.Em8.ControlNodes".citiMap.PMC.Machining_Assembly.IncrGood_Count AND NOT "Unit1.Em8.ControlNodes".citiMap.PMC.Machining_Assembly.IncrReject_Count);
   #_w2 := #_w1 AND NOT #citi_Ptrig[5];   // rising edge
   #citi_Ptrig[5] := #_w1;
   "Unit1.Em8.ControlNodes".citiMap.PMC.Machining_Assembly.Cycle_Time_Ready := (#_w2 OR "Unit1.Em8.ControlNodes".citiMap.PMC.Machining_Assembly.Cycle_Time_Ready) AND NOT #citiTon[5].Q;
   #citiTon[5].TON(IN := "Unit1.Em8.ControlNodes".citiMap.PMC.Machining_Assembly.Cycle_Time_Ready, PT := #citi);
END_REGION

REGION Network 133: Fault bit Level1 6
   RUNG wire#powerrail
      Contact( "Unit1.Em8.InstProDiag".State.C1 )
      wire#w1
      Coil( "Unit1.Em8.ControlNodes".citiMap.PMC.Machining_Assembly.Machine_FaultedLevel1 )
   END_RUNG
   RUNG wire#powerrail
      Contact( #citiTest[6] )
   END_RUNG wire#w1
   // the same network as SCL:
   "Unit1.Em8.ControlNodes".citiMap.PMC.Machining_Assembly.Machine_FaultedLevel1 := "Unit1.Em8.InstProDiag".State.C1 OR #citiTest[6];
END_REGION

REGION Network 134: Fault bit Level2 7
   RUNG wire#powerrail
      Contact( "Unit1.Em8.InstProDiag".State.C2 )
      wire#w1
      Coil( "Unit1.Em8.ControlNodes".citiMap.PMC.Machining_Assembly.Machine_FaultedLevel2 )
   END_RUNG
   RUNG wire#powerrail
      Contact( #citiTest[7] )
   END_RUNG wire#w1
   // the same network as SCL:
   "Unit1.Em8.ControlNodes".citiMap.PMC.Machining_Assembly.Machine_FaultedLevel2 := "Unit1.Em8.InstProDiag".State.C2 OR #citiTest[7];
END_REGION

REGION Network 135: Pun 9
   RUNG wire#powerrail
      Contact( #citiTest[9] )
      P_Trig( #citi_Ptrig[9] )
      Coil( "Unit1.Em8.ControlNodes".citiMap.PMC.Machining_Assembly.PUNData_command )
   END_RUNG
   // the same network as SCL:
   #_w1 := #citiTest[9] AND NOT #citi_Ptrig[9];   // rising edge
   #citi_Ptrig[9] := #citiTest[9];
   "Unit1.Em8.ControlNodes".citiMap.PMC.Machining_Assembly.PUNData_command := #_w1;
END_REGION

REGION Network 137: ******************** PFE Events ********************
END_REGION

REGION Network 138: PFE Events
   // Call the PFE events according to GM specification or use cases
   RUNG wire#powerrail
      #instEventsPFE()
   END_RUNG
   // the same network as SCL:
   #instEventsPFE();   // "Unit1.Em8.EventsPFE"
END_REGION

REGION Network 139: PFE Events Recipe
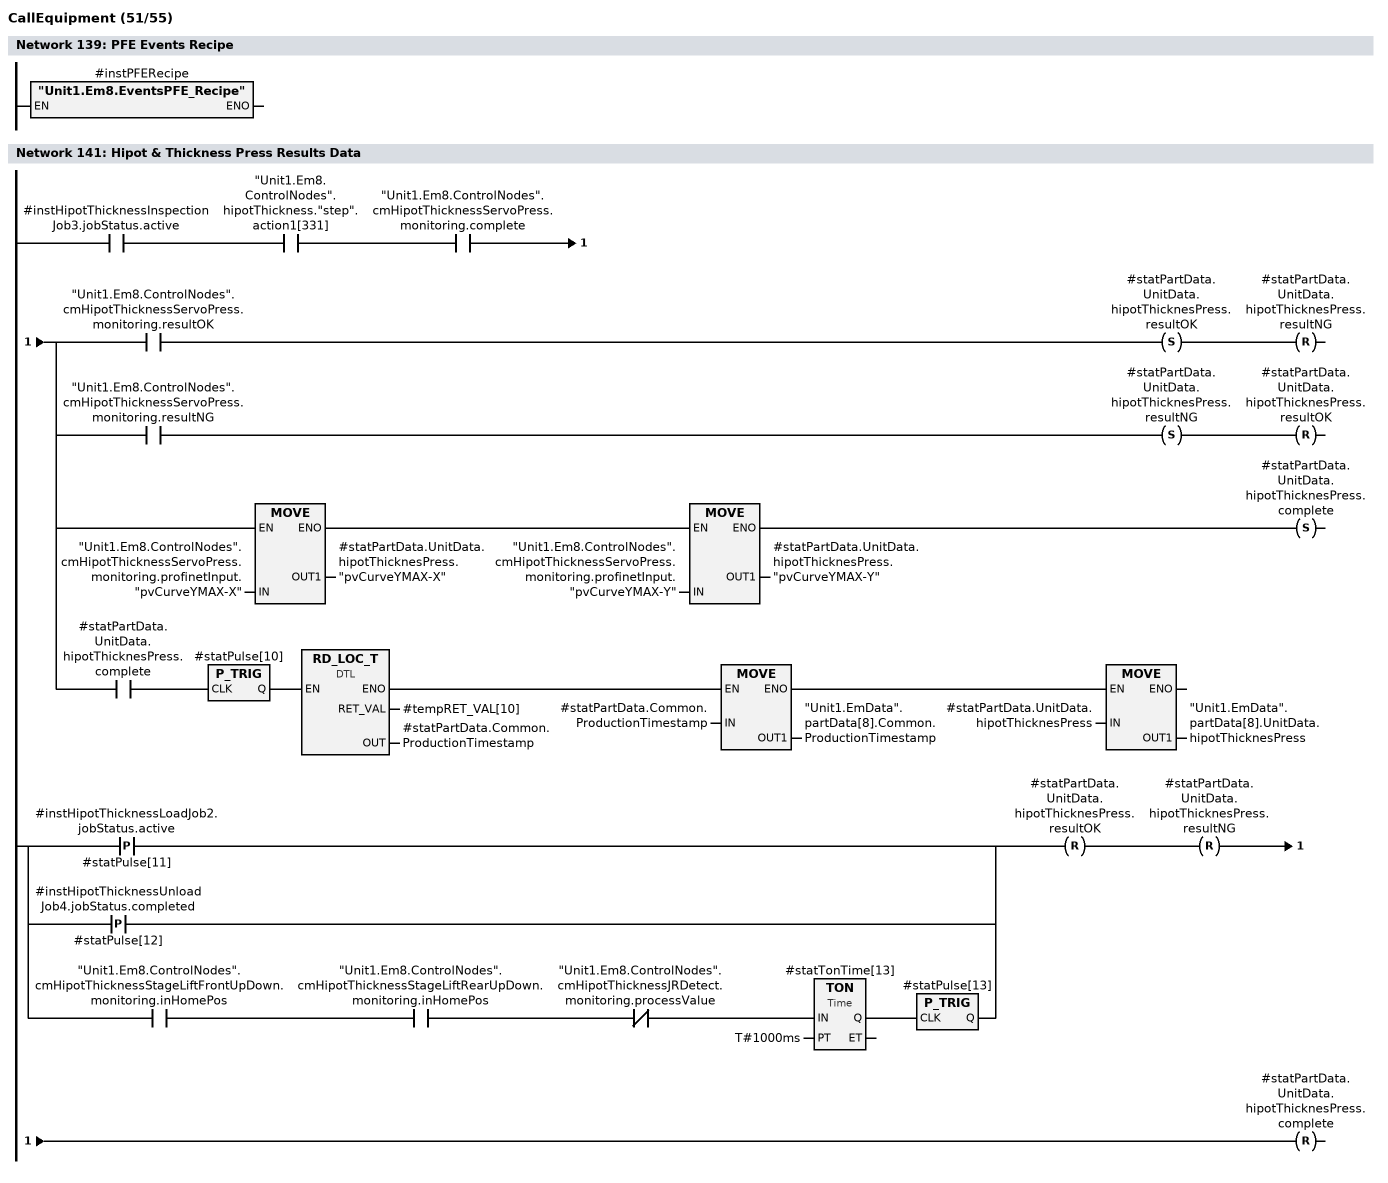
   RUNG wire#powerrail
      #instPFERecipe()
   END_RUNG
   // the same network as SCL:
   #instPFERecipe();   // "Unit1.Em8.EventsPFE_Recipe"
END_REGION

REGION Network 140: ************************ Part Results Data ************************
END_REGION

REGION Network 141: Hipot & Thickness Press Results Data
   RUNG wire#powerrail
      Contact( #instHipotThicknessInspectionJob3.jobStatus.active )
      Contact( "Unit1.Em8.ControlNodes".hipotThickness."step".action1[331] )
      Contact( "Unit1.Em8.ControlNodes".cmHipotThicknessServoPress.monitoring.complete )
      wire#w1
      Contact( "Unit1.Em8.ControlNodes".cmHipotThicknessServoPress.monitoring.resultOK )
      S_Coil( #statPartData.UnitData.hipotThicknesPress.resultOK )
      R_Coil( #statPartData.UnitData.hipotThicknesPress.resultNG )
   END_RUNG
   RUNG wire#w1
      Contact( "Unit1.Em8.ControlNodes".cmHipotThicknessServoPress.monitoring.resultNG )
      S_Coil( #statPartData.UnitData.hipotThicknesPress.resultNG )
      R_Coil( #statPartData.UnitData.hipotThicknesPress.resultOK )
   END_RUNG
   RUNG wire#w1
      Move(in := "Unit1.Em8.ControlNodes".cmHipotThicknessServoPress.monitoring.profinetInput."pvCurveYMAX-X", out1 => #statPartData.UnitData.hipotThicknesPress."pvCurveYMAX-X")
      Move(in := "Unit1.Em8.ControlNodes".cmHipotThicknessServoPress.monitoring.profinetInput."pvCurveYMAX-Y", out1 => #statPartData.UnitData.hipotThicknesPress."pvCurveYMAX-Y")
      S_Coil( #statPartData.UnitData.hipotThicknesPress.complete )
   END_RUNG
   RUNG wire#w1
      Contact( #statPartData.UnitData.hipotThicknesPress.complete )
      P_Trig( #statPulse[10] )
      { S7_Templates := "date_type := DTL" } RD_LOC_T(RET_VAL => #tempRET_VAL[10], OUT => #statPartData.Common.ProductionTimestamp)
      Move(in := #statPartData.Common.ProductionTimestamp, out1 => "Unit1.EmData".partData[8].Common.ProductionTimestamp)
      Move(in := #statPartData.UnitData.hipotThicknesPress, out1 => "Unit1.EmData".partData[8].UnitData.hipotThicknesPress)
   END_RUNG
   RUNG wire#powerrail
      P_Contact(operand := #instHipotThicknessLoadJob2.jobStatus.active, bit := #statPulse[11])
      wire#w2
      R_Coil( #statPartData.UnitData.hipotThicknesPress.resultOK )
      R_Coil( #statPartData.UnitData.hipotThicknesPress.resultNG )
      R_Coil( #statPartData.UnitData.hipotThicknesPress.complete )
   END_RUNG
   RUNG wire#powerrail
      P_Contact(operand := #instHipotThicknessUnloadJob4.jobStatus.completed, bit := #statPulse[12])
   END_RUNG wire#w2
   RUNG wire#powerrail
      Contact( "Unit1.Em8.ControlNodes".cmHipotThicknessStageLiftFrontUpDown.monitoring.inHomePos )
      Contact( "Unit1.Em8.ControlNodes".cmHipotThicknessStageLiftRearUpDown.monitoring.inHomePos )
      I_Contact( "Unit1.Em8.ControlNodes".cmHipotThicknessJRDetect.monitoring.processValue )
      { S7_Templates := "time_type := Time" } #statTonTime[13].TON(pt := T#1000ms, et =>)
      P_Trig( #statPulse[13] )
   END_RUNG wire#w2
   // the same network as SCL:
   #_w1 := #instHipotThicknessInspectionJob3.jobStatus.active AND "Unit1.Em8.ControlNodes".hipotThickness."step".action1[331] AND "Unit1.Em8.ControlNodes".cmHipotThicknessServoPress.monitoring.complete;
   IF #_w1 AND "Unit1.Em8.ControlNodes".cmHipotThicknessServoPress.monitoring.resultOK THEN
       #statPartData.UnitData.hipotThicknesPress.resultOK := TRUE;
       #statPartData.UnitData.hipotThicknesPress.resultNG := FALSE;
   END_IF;
   IF #_w1 AND "Unit1.Em8.ControlNodes".cmHipotThicknessServoPress.monitoring.resultNG THEN
       #statPartData.UnitData.hipotThicknesPress.resultNG := TRUE;
       #statPartData.UnitData.hipotThicknesPress.resultOK := FALSE;
   END_IF;
   IF #_w1 THEN
       #statPartData.UnitData.hipotThicknesPress."pvCurveYMAX-X" := "Unit1.Em8.ControlNodes".cmHipotThicknessServoPress.monitoring.profinetInput."pvCurveYMAX-X";
       #statPartData.UnitData.hipotThicknesPress."pvCurveYMAX-Y" := "Unit1.Em8.ControlNodes".cmHipotThicknessServoPress.monitoring.profinetInput."pvCurveYMAX-Y";
       #statPartData.UnitData.hipotThicknesPress.complete := TRUE;
   END_IF;
   #_w2 := #_w1 AND #statPartData.UnitData.hipotThicknesPress.complete;
   #_w3 := #_w2 AND NOT #statPulse[10];   // rising edge
   #statPulse[10] := #_w2;
   #tempRET_VAL[10] := RD_LOC_T(EN := #_w3, OUT => #statPartData.Common.ProductionTimestamp, ENO => #_w4);
   IF #_w4 THEN
       "Unit1.EmData".partData[8].Common.ProductionTimestamp := #statPartData.Common.ProductionTimestamp;
       "Unit1.EmData".partData[8].UnitData.hipotThicknesPress := #statPartData.UnitData.hipotThicknesPress;
   END_IF;
   #_w5 := #instHipotThicknessLoadJob2.jobStatus.active AND NOT #statPulse[11];   // rising edge of #instHipotThicknessLoadJob2.jobStatus.active
   #statPulse[11] := #instHipotThicknessLoadJob2.jobStatus.active;
   #_w6 := #instHipotThicknessUnloadJob4.jobStatus.completed AND NOT #statPulse[12];   // rising edge of #instHipotThicknessUnloadJob4.jobStatus.completed
   #statPulse[12] := #instHipotThicknessUnloadJob4.jobStatus.completed;
   #statTonTime[13].TON(IN := "Unit1.Em8.ControlNodes".cmHipotThicknessStageLiftFrontUpDown.monitoring.inHomePos AND "Unit1.Em8.ControlNodes".cmHipotThicknessStageLiftRearUpDown.monitoring.inHomePos AND NOT "Unit1.Em8.ControlNodes".cmHipotThicknessJRDetect.monitoring.processValue,
                        PT := T#1000ms);
   #_w7 := #statTonTime[13].Q AND NOT #statPulse[13];   // rising edge
   #statPulse[13] := #statTonTime[13].Q;
   IF #_w5 OR #_w6 OR #_w7 THEN
       #statPartData.UnitData.hipotThicknesPress.resultOK := FALSE;
       #statPartData.UnitData.hipotThicknesPress.resultNG := FALSE;
       #statPartData.UnitData.hipotThicknesPress.complete := FALSE;
   END_IF;
END_REGION

REGION Network 142: Thickness Results Data
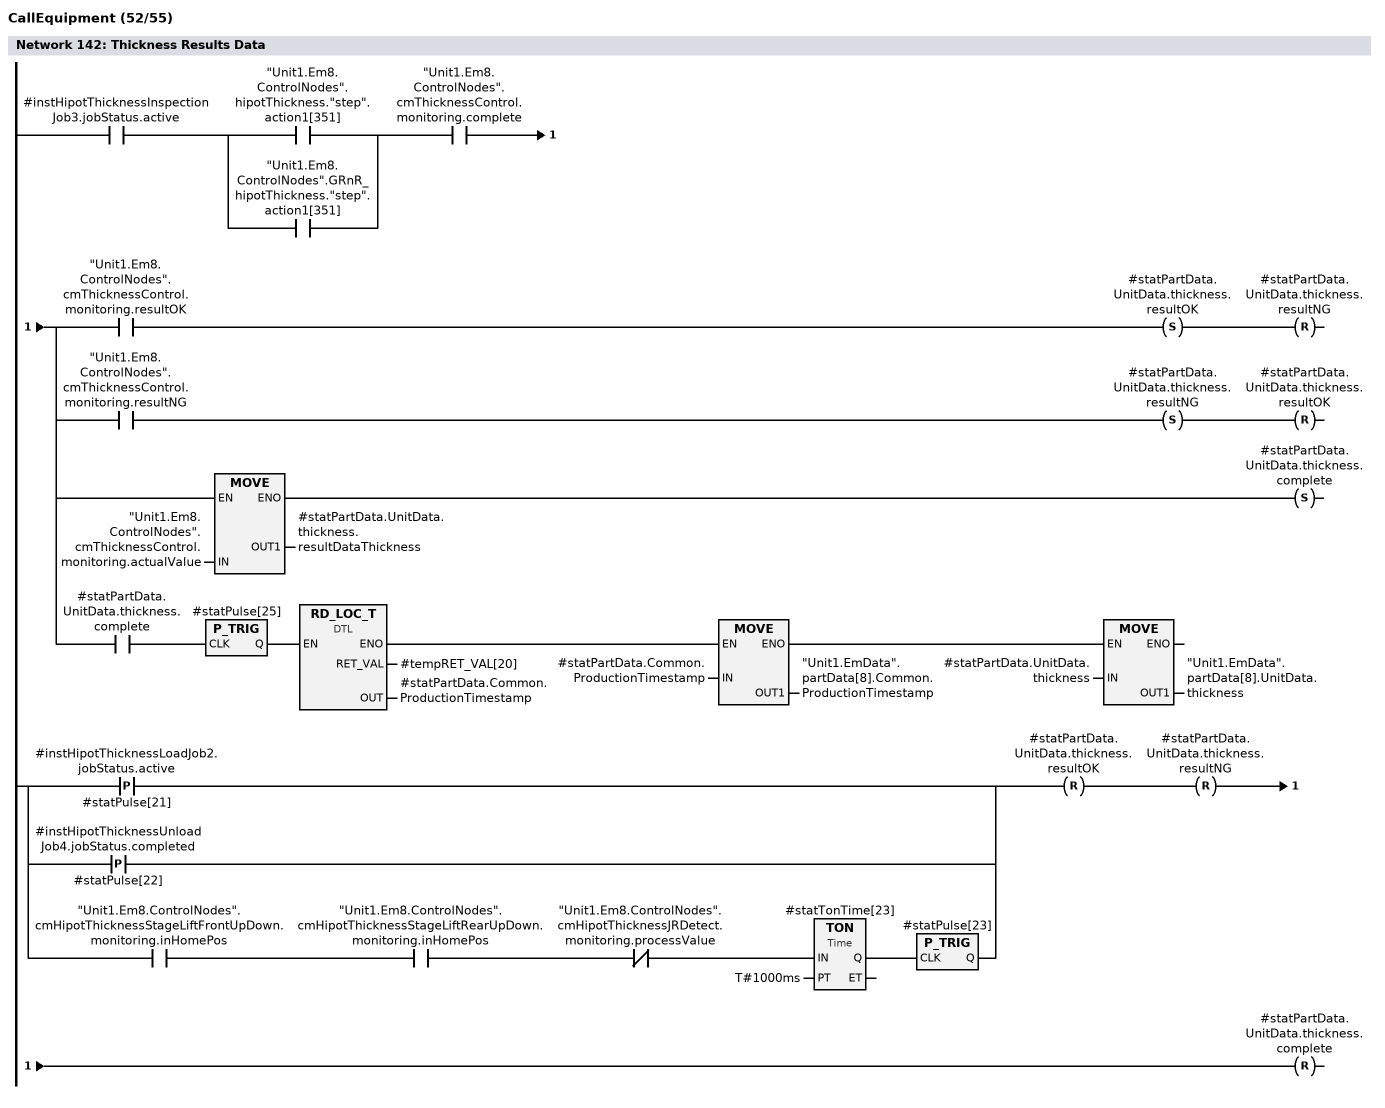
   RUNG wire#powerrail
      Contact( #instHipotThicknessInspectionJob3.jobStatus.active )
      wire#w1
      Contact( "Unit1.Em8.ControlNodes".hipotThickness."step".action1[351] )
      wire#w2
      Contact( "Unit1.Em8.ControlNodes".cmThicknessControl.monitoring.complete )
      wire#w3
      Contact( "Unit1.Em8.ControlNodes".cmThicknessControl.monitoring.resultOK )
      S_Coil( #statPartData.UnitData.thickness.resultOK )
      R_Coil( #statPartData.UnitData.thickness.resultNG )
   END_RUNG
   RUNG wire#w1
      Contact( "Unit1.Em8.ControlNodes".GRnR_hipotThickness."step".action1[351] )
   END_RUNG wire#w2
   RUNG wire#w3
      Contact( "Unit1.Em8.ControlNodes".cmThicknessControl.monitoring.resultNG )
      S_Coil( #statPartData.UnitData.thickness.resultNG )
      R_Coil( #statPartData.UnitData.thickness.resultOK )
   END_RUNG
   RUNG wire#w3
      Move(in := "Unit1.Em8.ControlNodes".cmThicknessControl.monitoring.actualValue, out1 => #statPartData.UnitData.thickness.resultDataThickness)
      S_Coil( #statPartData.UnitData.thickness.complete )
   END_RUNG
   RUNG wire#w3
      Contact( #statPartData.UnitData.thickness.complete )
      P_Trig( #statPulse[25] )
      { S7_Templates := "date_type := DTL" } RD_LOC_T(RET_VAL => #tempRET_VAL[20], OUT => #statPartData.Common.ProductionTimestamp)
      Move(in := #statPartData.Common.ProductionTimestamp, out1 => "Unit1.EmData".partData[8].Common.ProductionTimestamp)
      Move(in := #statPartData.UnitData.thickness, out1 => "Unit1.EmData".partData[8].UnitData.thickness)
   END_RUNG
   RUNG wire#powerrail
      P_Contact(operand := #instHipotThicknessLoadJob2.jobStatus.active, bit := #statPulse[21])
      wire#w4
      R_Coil( #statPartData.UnitData.thickness.resultOK )
      R_Coil( #statPartData.UnitData.thickness.resultNG )
      R_Coil( #statPartData.UnitData.thickness.complete )
   END_RUNG
   RUNG wire#powerrail
      P_Contact(operand := #instHipotThicknessUnloadJob4.jobStatus.completed, bit := #statPulse[22])
   END_RUNG wire#w4
   RUNG wire#powerrail
      Contact( "Unit1.Em8.ControlNodes".cmHipotThicknessStageLiftFrontUpDown.monitoring.inHomePos )
      Contact( "Unit1.Em8.ControlNodes".cmHipotThicknessStageLiftRearUpDown.monitoring.inHomePos )
      I_Contact( "Unit1.Em8.ControlNodes".cmHipotThicknessJRDetect.monitoring.processValue )
      { S7_Templates := "time_type := Time" } #statTonTime[23].TON(pt := T#1000ms, et =>)
      P_Trig( #statPulse[23] )
   END_RUNG wire#w4
   // the same network as SCL:
   #_w1 := #instHipotThicknessInspectionJob3.jobStatus.active AND ("Unit1.Em8.ControlNodes".hipotThickness."step".action1[351] OR "Unit1.Em8.ControlNodes".GRnR_hipotThickness."step".action1[351]) AND "Unit1.Em8.ControlNodes".cmThicknessControl.monitoring.complete;
   IF #_w1 AND "Unit1.Em8.ControlNodes".cmThicknessControl.monitoring.resultOK THEN
       #statPartData.UnitData.thickness.resultOK := TRUE;
       #statPartData.UnitData.thickness.resultNG := FALSE;
   END_IF;
   IF #_w1 AND "Unit1.Em8.ControlNodes".cmThicknessControl.monitoring.resultNG THEN
       #statPartData.UnitData.thickness.resultNG := TRUE;
       #statPartData.UnitData.thickness.resultOK := FALSE;
   END_IF;
   IF #_w1 THEN
       #statPartData.UnitData.thickness.resultDataThickness := "Unit1.Em8.ControlNodes".cmThicknessControl.monitoring.actualValue;
       #statPartData.UnitData.thickness.complete := TRUE;
   END_IF;
   #_w2 := #_w1 AND #statPartData.UnitData.thickness.complete;
   #_w3 := #_w2 AND NOT #statPulse[25];   // rising edge
   #statPulse[25] := #_w2;
   #tempRET_VAL[20] := RD_LOC_T(EN := #_w3, OUT => #statPartData.Common.ProductionTimestamp, ENO => #_w4);
   IF #_w4 THEN
       "Unit1.EmData".partData[8].Common.ProductionTimestamp := #statPartData.Common.ProductionTimestamp;
       "Unit1.EmData".partData[8].UnitData.thickness := #statPartData.UnitData.thickness;
   END_IF;
   #_w5 := #instHipotThicknessLoadJob2.jobStatus.active AND NOT #statPulse[21];   // rising edge of #instHipotThicknessLoadJob2.jobStatus.active
   #statPulse[21] := #instHipotThicknessLoadJob2.jobStatus.active;
   #_w6 := #instHipotThicknessUnloadJob4.jobStatus.completed AND NOT #statPulse[22];   // rising edge of #instHipotThicknessUnloadJob4.jobStatus.completed
   #statPulse[22] := #instHipotThicknessUnloadJob4.jobStatus.completed;
   #statTonTime[23].TON(IN := "Unit1.Em8.ControlNodes".cmHipotThicknessStageLiftFrontUpDown.monitoring.inHomePos AND "Unit1.Em8.ControlNodes".cmHipotThicknessStageLiftRearUpDown.monitoring.inHomePos AND NOT "Unit1.Em8.ControlNodes".cmHipotThicknessJRDetect.monitoring.processValue,
                        PT := T#1000ms);
   #_w7 := #statTonTime[23].Q AND NOT #statPulse[23];   // rising edge
   #statPulse[23] := #statTonTime[23].Q;
   IF #_w5 OR #_w6 OR #_w7 THEN
       #statPartData.UnitData.thickness.resultOK := FALSE;
       #statPartData.UnitData.thickness.resultNG := FALSE;
       #statPartData.UnitData.thickness.complete := FALSE;
   END_IF;
END_REGION

REGION Network 143: Hipot Results Data
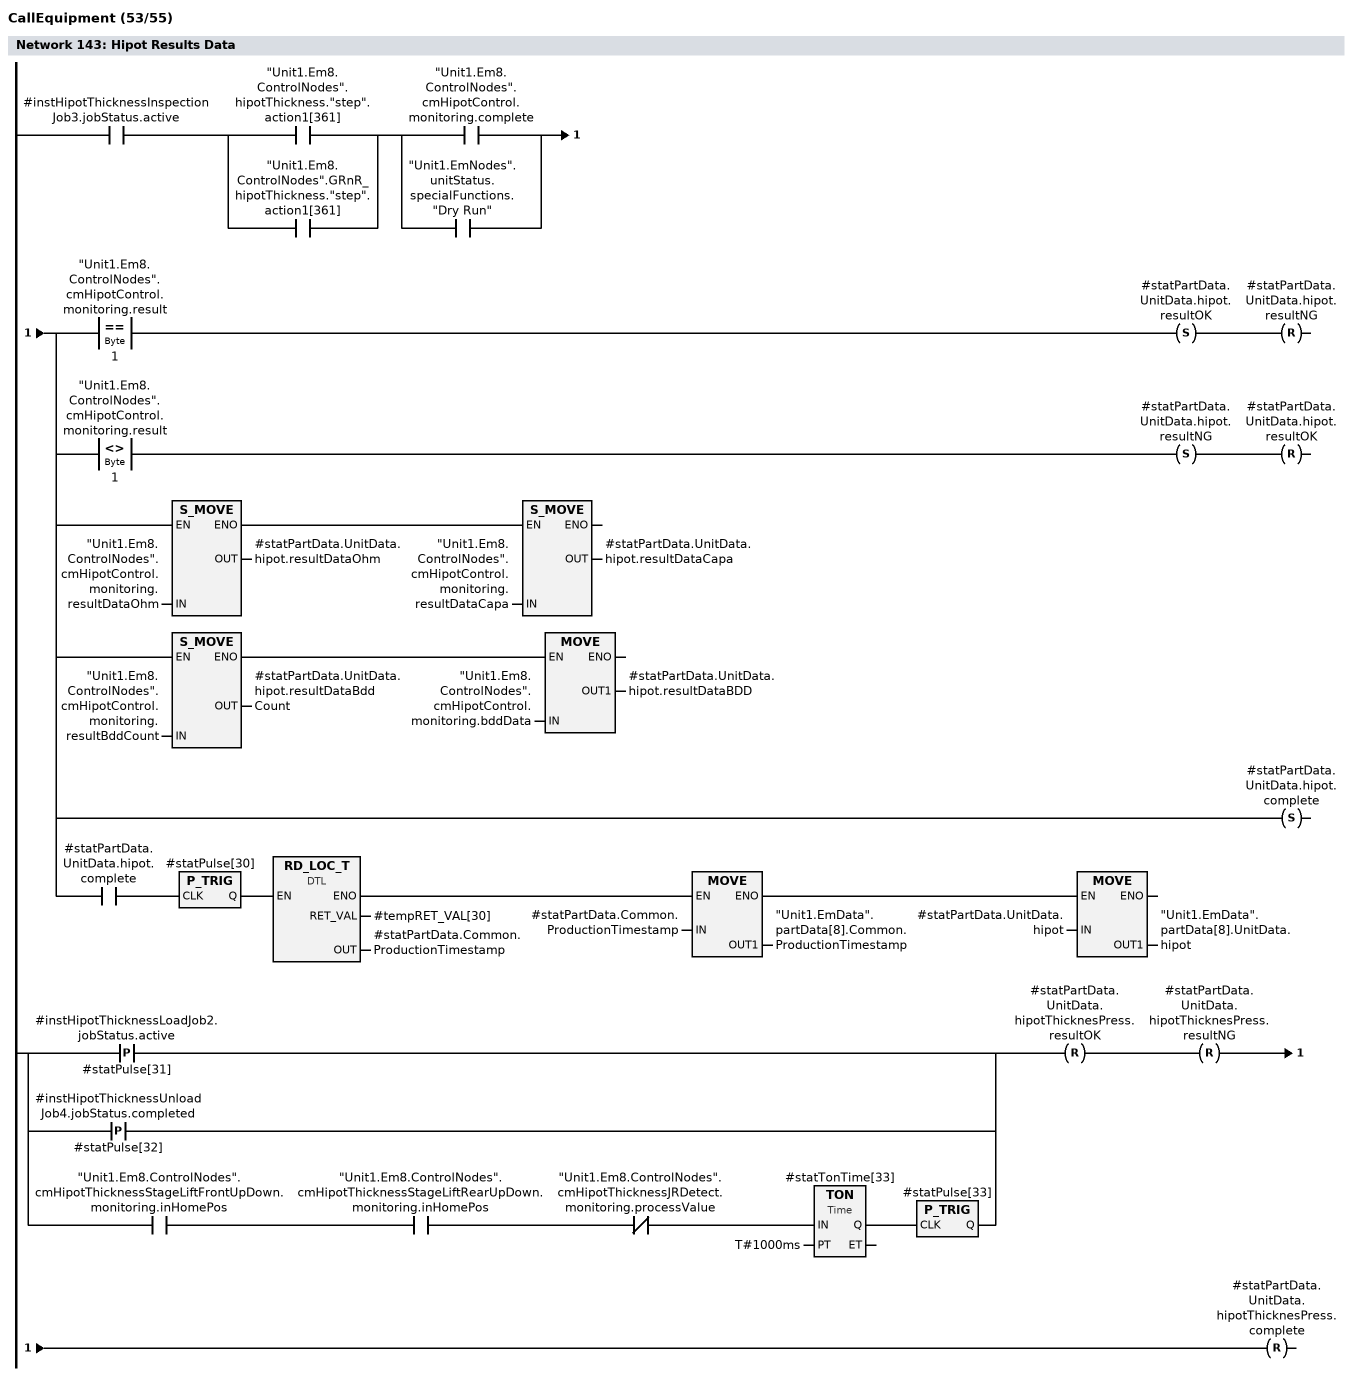
   RUNG wire#powerrail
      Contact( #instHipotThicknessInspectionJob3.jobStatus.active )
      wire#w1
      Contact( "Unit1.Em8.ControlNodes".hipotThickness."step".action1[361] )
      wire#w2
      Contact( "Unit1.Em8.ControlNodes".cmHipotControl.monitoring.complete )
      wire#w3
      { S7_Templates := "SrcType := Byte" } EQ_Contact(in1 := "Unit1.Em8.ControlNodes".cmHipotControl.monitoring.result, in2 := 1)
      S_Coil( #statPartData.UnitData.hipot.resultOK )
      R_Coil( #statPartData.UnitData.hipot.resultNG )
   END_RUNG
   RUNG wire#w1
      Contact( "Unit1.Em8.ControlNodes".GRnR_hipotThickness."step".action1[361] )
   END_RUNG wire#w2
   RUNG wire#w2
      Contact( "Unit1.EmNodes".unitStatus.specialFunctions."Dry Run" )
   END_RUNG wire#w3
   RUNG wire#w3
      { S7_Templates := "SrcType := Byte" } NE_Contact(in1 := "Unit1.Em8.ControlNodes".cmHipotControl.monitoring.result, in2 := 1)
      S_Coil( #statPartData.UnitData.hipot.resultNG )
      R_Coil( #statPartData.UnitData.hipot.resultOK )
   END_RUNG
   RUNG wire#w3
      S_Move(in := "Unit1.Em8.ControlNodes".cmHipotControl.monitoring.resultDataOhm, out => #statPartData.UnitData.hipot.resultDataOhm)
      S_Move(in := "Unit1.Em8.ControlNodes".cmHipotControl.monitoring.resultDataCapa, out => #statPartData.UnitData.hipot.resultDataCapa)
   END_RUNG
   RUNG wire#w3
      S_Move(in := "Unit1.Em8.ControlNodes".cmHipotControl.monitoring.resultBddCount, out => #statPartData.UnitData.hipot.resultDataBddCount)
      Move(in := "Unit1.Em8.ControlNodes".cmHipotControl.monitoring.bddData, out1 => #statPartData.UnitData.hipot.resultDataBDD)
   END_RUNG
   RUNG wire#w3
      S_Coil( #statPartData.UnitData.hipot.complete )
   END_RUNG
   RUNG wire#w3
      Contact( #statPartData.UnitData.hipot.complete )
      P_Trig( #statPulse[30] )
      { S7_Templates := "date_type := DTL" } RD_LOC_T(RET_VAL => #tempRET_VAL[30], OUT => #statPartData.Common.ProductionTimestamp)
      Move(in := #statPartData.Common.ProductionTimestamp, out1 => "Unit1.EmData".partData[8].Common.ProductionTimestamp)
      Move(in := #statPartData.UnitData.hipot, out1 => "Unit1.EmData".partData[8].UnitData.hipot)
   END_RUNG
   RUNG wire#powerrail
      P_Contact(operand := #instHipotThicknessLoadJob2.jobStatus.active, bit := #statPulse[31])
      wire#w4
      R_Coil( #statPartData.UnitData.hipotThicknesPress.resultOK )
      R_Coil( #statPartData.UnitData.hipotThicknesPress.resultNG )
      R_Coil( #statPartData.UnitData.hipotThicknesPress.complete )
   END_RUNG
   RUNG wire#powerrail
      P_Contact(operand := #instHipotThicknessUnloadJob4.jobStatus.completed, bit := #statPulse[32])
   END_RUNG wire#w4
   RUNG wire#powerrail
      Contact( "Unit1.Em8.ControlNodes".cmHipotThicknessStageLiftFrontUpDown.monitoring.inHomePos )
      Contact( "Unit1.Em8.ControlNodes".cmHipotThicknessStageLiftRearUpDown.monitoring.inHomePos )
      I_Contact( "Unit1.Em8.ControlNodes".cmHipotThicknessJRDetect.monitoring.processValue )
      { S7_Templates := "time_type := Time" } #statTonTime[33].TON(pt := T#1000ms, et =>)
      P_Trig( #statPulse[33] )
   END_RUNG wire#w4
   // the same network as SCL:
   #_w1 := #instHipotThicknessInspectionJob3.jobStatus.active AND ("Unit1.Em8.ControlNodes".hipotThickness."step".action1[361] OR "Unit1.Em8.ControlNodes".GRnR_hipotThickness."step".action1[361]) AND ("Unit1.Em8.ControlNodes".cmHipotControl.monitoring.complete OR "Unit1.EmNodes".unitStatus.specialFunctions."Dry Run");
   IF #_w1 AND ("Unit1.Em8.ControlNodes".cmHipotControl.monitoring.result = 1) THEN
       #statPartData.UnitData.hipot.resultOK := TRUE;
       #statPartData.UnitData.hipot.resultNG := FALSE;
   END_IF;
   IF #_w1 AND ("Unit1.Em8.ControlNodes".cmHipotControl.monitoring.result <> 1) THEN
       #statPartData.UnitData.hipot.resultNG := TRUE;
       #statPartData.UnitData.hipot.resultOK := FALSE;
   END_IF;
   IF #_w1 THEN
       #statPartData.UnitData.hipot.resultDataOhm := "Unit1.Em8.ControlNodes".cmHipotControl.monitoring.resultDataOhm;
       #statPartData.UnitData.hipot.resultDataCapa := "Unit1.Em8.ControlNodes".cmHipotControl.monitoring.resultDataCapa;
       #statPartData.UnitData.hipot.resultDataBddCount := "Unit1.Em8.ControlNodes".cmHipotControl.monitoring.resultBddCount;
       #statPartData.UnitData.hipot.resultDataBDD := "Unit1.Em8.ControlNodes".cmHipotControl.monitoring.bddData;
       #statPartData.UnitData.hipot.complete := TRUE;
   END_IF;
   #_w2 := #_w1 AND #statPartData.UnitData.hipot.complete;
   #_w3 := #_w2 AND NOT #statPulse[30];   // rising edge
   #statPulse[30] := #_w2;
   #tempRET_VAL[30] := RD_LOC_T(EN := #_w3, OUT => #statPartData.Common.ProductionTimestamp, ENO => #_w4);
   IF #_w4 THEN
       "Unit1.EmData".partData[8].Common.ProductionTimestamp := #statPartData.Common.ProductionTimestamp;
       "Unit1.EmData".partData[8].UnitData.hipot := #statPartData.UnitData.hipot;
   END_IF;
   #_w5 := #instHipotThicknessLoadJob2.jobStatus.active AND NOT #statPulse[31];   // rising edge of #instHipotThicknessLoadJob2.jobStatus.active
   #statPulse[31] := #instHipotThicknessLoadJob2.jobStatus.active;
   #_w6 := #instHipotThicknessUnloadJob4.jobStatus.completed AND NOT #statPulse[32];   // rising edge of #instHipotThicknessUnloadJob4.jobStatus.completed
   #statPulse[32] := #instHipotThicknessUnloadJob4.jobStatus.completed;
   #statTonTime[33].TON(IN := "Unit1.Em8.ControlNodes".cmHipotThicknessStageLiftFrontUpDown.monitoring.inHomePos AND "Unit1.Em8.ControlNodes".cmHipotThicknessStageLiftRearUpDown.monitoring.inHomePos AND NOT "Unit1.Em8.ControlNodes".cmHipotThicknessJRDetect.monitoring.processValue,
                        PT := T#1000ms);
   #_w7 := #statTonTime[33].Q AND NOT #statPulse[33];   // rising edge
   #statPulse[33] := #statTonTime[33].Q;
   IF #_w5 OR #_w6 OR #_w7 THEN
       #statPartData.UnitData.hipotThicknesPress.resultOK := FALSE;
       #statPartData.UnitData.hipotThicknesPress.resultNG := FALSE;
       #statPartData.UnitData.hipotThicknesPress.complete := FALSE;
   END_IF;
END_REGION

REGION Network 145: ******************** Unit Output ********************
END_REGION

REGION Network 146: EM08 Relations Em Linked Status
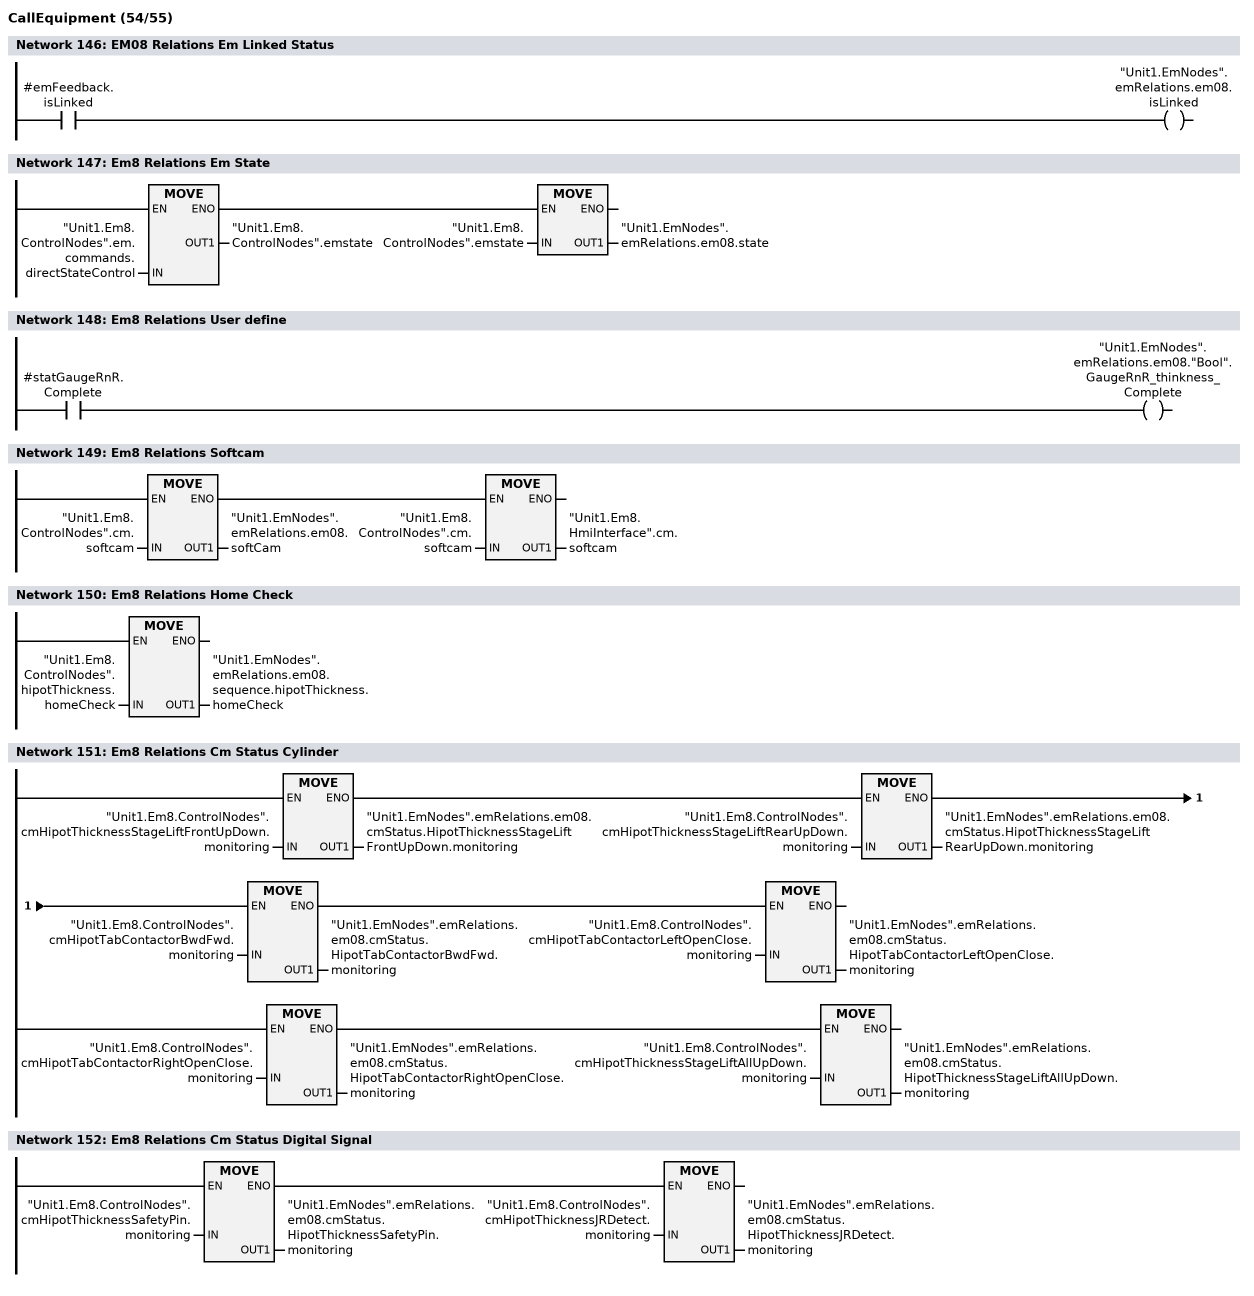
   RUNG wire#powerrail
      Contact( #emFeedback.isLinked )
      Coil( "Unit1.EmNodes".emRelations.em08.isLinked )
   END_RUNG
   // the same network as SCL:
   "Unit1.EmNodes".emRelations.em08.isLinked := #emFeedback.isLinked;
END_REGION

REGION Network 147: Em8 Relations Em State
   RUNG wire#powerrail
      Move(in := "Unit1.Em8.ControlNodes".em.commands.directStateControl, out1 => "Unit1.Em8.ControlNodes".emstate)
      Move(in := "Unit1.Em8.ControlNodes".emstate, out1 => "Unit1.EmNodes".emRelations.em08.state)
   END_RUNG
   // the same network as SCL:
   "Unit1.Em8.ControlNodes".emstate := "Unit1.Em8.ControlNodes".em.commands.directStateControl;
   "Unit1.EmNodes".emRelations.em08.state := "Unit1.Em8.ControlNodes".emstate;
END_REGION

REGION Network 148: Em8 Relations User define
   RUNG wire#powerrail
      Contact( #statGaugeRnR.Complete )
      Coil( "Unit1.EmNodes".emRelations.em08."Bool".GaugeRnR_thinkness_Complete )
   END_RUNG
   // the same network as SCL:
   "Unit1.EmNodes".emRelations.em08."Bool".GaugeRnR_thinkness_Complete := #statGaugeRnR.Complete;
END_REGION

REGION Network 149: Em8 Relations Softcam
   RUNG wire#powerrail
      Move(in := "Unit1.Em8.ControlNodes".cm.softcam, out1 => "Unit1.EmNodes".emRelations.em08.softCam)
      Move(in := "Unit1.Em8.ControlNodes".cm.softcam, out1 => "Unit1.Em8.HmiInterface".cm.softcam)
   END_RUNG
   // the same network as SCL:
   "Unit1.EmNodes".emRelations.em08.softCam := "Unit1.Em8.ControlNodes".cm.softcam;
   "Unit1.Em8.HmiInterface".cm.softcam := "Unit1.Em8.ControlNodes".cm.softcam;
END_REGION

REGION Network 150: Em8 Relations Home Check
   RUNG wire#powerrail
      Move(in := "Unit1.Em8.ControlNodes".hipotThickness.homeCheck, out1 => "Unit1.EmNodes".emRelations.em08.sequence.hipotThickness.homeCheck)
   END_RUNG
   // the same network as SCL:
   "Unit1.EmNodes".emRelations.em08.sequence.hipotThickness.homeCheck := "Unit1.Em8.ControlNodes".hipotThickness.homeCheck;
END_REGION

REGION Network 151: Em8 Relations Cm Status Cylinder
   RUNG wire#powerrail
      Move(in := "Unit1.Em8.ControlNodes".cmHipotThicknessStageLiftFrontUpDown.monitoring, out1 => "Unit1.EmNodes".emRelations.em08.cmStatus.HipotThicknessStageLiftFrontUpDown.monitoring)
      Move(in := "Unit1.Em8.ControlNodes".cmHipotThicknessStageLiftRearUpDown.monitoring, out1 => "Unit1.EmNodes".emRelations.em08.cmStatus.HipotThicknessStageLiftRearUpDown.monitoring)
      Move(in := "Unit1.Em8.ControlNodes".cmHipotTabContactorBwdFwd.monitoring, out1 => "Unit1.EmNodes".emRelations.em08.cmStatus.HipotTabContactorBwdFwd.monitoring)
      Move(in := "Unit1.Em8.ControlNodes".cmHipotTabContactorLeftOpenClose.monitoring, out1 => "Unit1.EmNodes".emRelations.em08.cmStatus.HipotTabContactorLeftOpenClose.monitoring)
   END_RUNG
   RUNG wire#powerrail
      Move(in := "Unit1.Em8.ControlNodes".cmHipotTabContactorRightOpenClose.monitoring, out1 => "Unit1.EmNodes".emRelations.em08.cmStatus.HipotTabContactorRightOpenClose.monitoring)
      Move(in := "Unit1.Em8.ControlNodes".cmHipotThicknessStageLiftAllUpDown.monitoring, out1 => "Unit1.EmNodes".emRelations.em08.cmStatus.HipotThicknessStageLiftAllUpDown.monitoring)
   END_RUNG
   // the same network as SCL:
   "Unit1.EmNodes".emRelations.em08.cmStatus.HipotThicknessStageLiftFrontUpDown.monitoring := "Unit1.Em8.ControlNodes".cmHipotThicknessStageLiftFrontUpDown.monitoring;
   "Unit1.EmNodes".emRelations.em08.cmStatus.HipotThicknessStageLiftRearUpDown.monitoring := "Unit1.Em8.ControlNodes".cmHipotThicknessStageLiftRearUpDown.monitoring;
   "Unit1.EmNodes".emRelations.em08.cmStatus.HipotTabContactorBwdFwd.monitoring := "Unit1.Em8.ControlNodes".cmHipotTabContactorBwdFwd.monitoring;
   "Unit1.EmNodes".emRelations.em08.cmStatus.HipotTabContactorLeftOpenClose.monitoring := "Unit1.Em8.ControlNodes".cmHipotTabContactorLeftOpenClose.monitoring;
   "Unit1.EmNodes".emRelations.em08.cmStatus.HipotTabContactorRightOpenClose.monitoring := "Unit1.Em8.ControlNodes".cmHipotTabContactorRightOpenClose.monitoring;
   "Unit1.EmNodes".emRelations.em08.cmStatus.HipotThicknessStageLiftAllUpDown.monitoring := "Unit1.Em8.ControlNodes".cmHipotThicknessStageLiftAllUpDown.monitoring;
END_REGION

REGION Network 152: Em8 Relations Cm Status Digital Signal
   RUNG wire#powerrail
      Move(in := "Unit1.Em8.ControlNodes".cmHipotThicknessSafetyPin.monitoring, out1 => "Unit1.EmNodes".emRelations.em08.cmStatus.HipotThicknessSafetyPin.monitoring)
      Move(in := "Unit1.Em8.ControlNodes".cmHipotThicknessJRDetect.monitoring, out1 => "Unit1.EmNodes".emRelations.em08.cmStatus.HipotThicknessJRDetect.monitoring)
   END_RUNG
   // the same network as SCL:
   "Unit1.EmNodes".emRelations.em08.cmStatus.HipotThicknessSafetyPin.monitoring := "Unit1.Em8.ControlNodes".cmHipotThicknessSafetyPin.monitoring;
   "Unit1.EmNodes".emRelations.em08.cmStatus.HipotThicknessJRDetect.monitoring := "Unit1.Em8.ControlNodes".cmHipotThicknessJRDetect.monitoring;
END_REGION

REGION Network 153
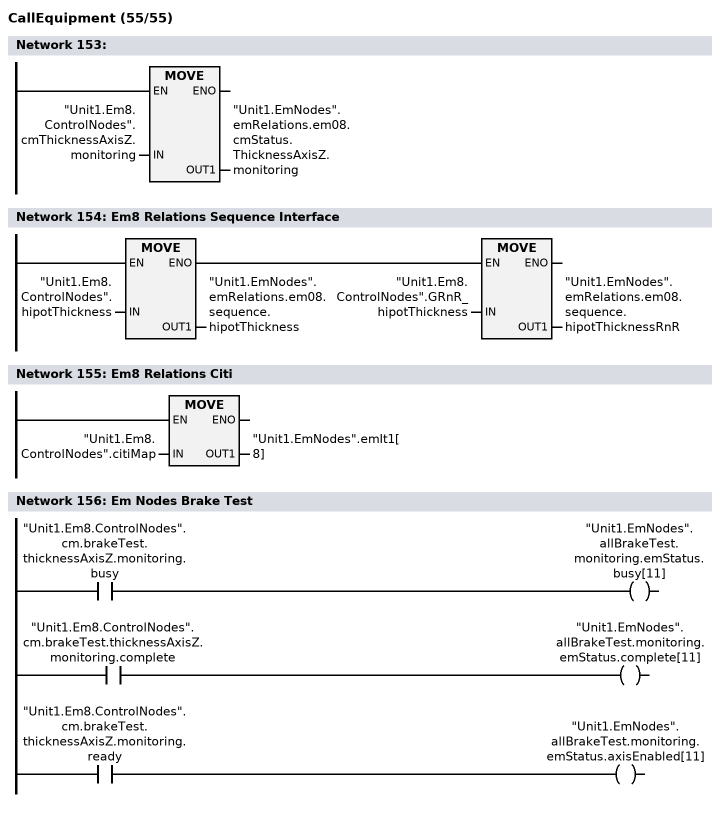
   RUNG wire#powerrail
      Move(in := "Unit1.Em8.ControlNodes".cmThicknessAxisZ.monitoring, out1 => "Unit1.EmNodes".emRelations.em08.cmStatus.ThicknessAxisZ.monitoring)
   END_RUNG
   // the same network as SCL:
   "Unit1.EmNodes".emRelations.em08.cmStatus.ThicknessAxisZ.monitoring := "Unit1.Em8.ControlNodes".cmThicknessAxisZ.monitoring;
END_REGION

REGION Network 154: Em8 Relations Sequence Interface
   RUNG wire#powerrail
      Move(in := "Unit1.Em8.ControlNodes".hipotThickness, out1 => "Unit1.EmNodes".emRelations.em08.sequence.hipotThickness)
      Move(in := "Unit1.Em8.ControlNodes".GRnR_hipotThickness, out1 => "Unit1.EmNodes".emRelations.em08.sequence.hipotThicknessRnR)
   END_RUNG
   // the same network as SCL:
   "Unit1.EmNodes".emRelations.em08.sequence.hipotThickness := "Unit1.Em8.ControlNodes".hipotThickness;
   "Unit1.EmNodes".emRelations.em08.sequence.hipotThicknessRnR := "Unit1.Em8.ControlNodes".GRnR_hipotThickness;
END_REGION

REGION Network 155: Em8 Relations Citi
   RUNG wire#powerrail
      Move(in := "Unit1.Em8.ControlNodes".citiMap, out1 => "Unit1.EmNodes".emIt1[8])
   END_RUNG
   // the same network as SCL:
   "Unit1.EmNodes".emIt1[8] := "Unit1.Em8.ControlNodes".citiMap;
END_REGION

REGION Network 156: Em Nodes Brake Test
   RUNG wire#powerrail
      Contact( "Unit1.Em8.ControlNodes".cm.brakeTest.thicknessAxisZ.monitoring.busy )
      Coil( "Unit1.EmNodes".allBrakeTest.monitoring.emStatus.busy[11] )
   END_RUNG
   RUNG wire#powerrail
      Contact( "Unit1.Em8.ControlNodes".cm.brakeTest.thicknessAxisZ.monitoring.complete )
      Coil( "Unit1.EmNodes".allBrakeTest.monitoring.emStatus.complete[11] )
   END_RUNG
   RUNG wire#powerrail
      Contact( "Unit1.Em8.ControlNodes".cm.brakeTest.thicknessAxisZ.monitoring.ready )
      Coil( "Unit1.EmNodes".allBrakeTest.monitoring.emStatus.axisEnabled[11] )
   END_RUNG
   // the same network as SCL:
   "Unit1.EmNodes".allBrakeTest.monitoring.emStatus.busy[11] := "Unit1.Em8.ControlNodes".cm.brakeTest.thicknessAxisZ.monitoring.busy;
   "Unit1.EmNodes".allBrakeTest.monitoring.emStatus.complete[11] := "Unit1.Em8.ControlNodes".cm.brakeTest.thicknessAxisZ.monitoring.complete;
   "Unit1.EmNodes".allBrakeTest.monitoring.emStatus.axisEnabled[11] := "Unit1.Em8.ControlNodes".cm.brakeTest.thicknessAxisZ.monitoring.ready;
END_REGION
END_FUNCTION_BLOCK
